    220: // Leak detection
      IF TRUE
      AND _m_LeakTest1_LeakDet()
			THEN 
        THIS^.stSeqCtrlGeneral.iInternalSeqStateCase := 230;
			END_IF
      
    230: // Stop and delay
      IF TRUE
      AND _m_Delay(DelayTime:= REAL_TO_TIME(THIS^.stLT1Params.rRestDelay * 1000))
      AND THIS^.itfCounterCyl.M_Stop()
			THEN 
        IF THIS^.bDoubleActing THEN
          THIS^.stSeqCtrlGeneral.iInternalSeqStateCase := 240; 
        ELSE
          THIS^.stSeqCtrlGeneral.iInternalSeqStateCase := 241; 
        END_IF
			END_IF
      
    240: // Move to Middle position
      IF TRUE
      AND THIS^.itfTestCyl.M_ToHP(ePressureType:= E_PRESSURE_TYPE.FORCE, 
                                  rWorkPressure:= THIS^.stLT1Params.rLoadForceB * 1000, 
                                  bPressureRegulation:= FALSE,
                                  eSpeedType:= E_SPEED_TYPE.PERCENT, 
                                  rSpeed:= 50)
      AND THIS^.itfCounterCyl.M_ToHP(ePressureType:= E_PRESSURE_TYPE.VALUE, 
                                     rWorkPressure:= 0, 
                                     bPressureRegulation:= FALSE,
                                     eSpeedType:= E_SPEED_TYPE.PERCENT, 
                                     rSpeed:= 50)
			THEN 
        IF THIS^.itfTestCyl.P_Position <= THIS^.itfTestCyl.P_StrokeLength / 2 THEN
				  THIS^.stSeqCtrlGeneral.iInternalSeqStateCase := 250; 
        END_IF
			END_IF
      
    241: // Move to Middle position
      IF TRUE
      AND THIS^.itfTestCyl.M_ToHP(ePressureType:= E_PRESSURE_TYPE.VALUE, 
                                  rWorkPressure:= 0, 
                                  bPressureRegulation:= FALSE,
                                  eSpeedType:= E_SPEED_TYPE.PERCENT, 
                                  rSpeed:= 50)
      AND THIS^.itfCounterCyl.M_ToWP(ePressureType:= E_PRESSURE_TYPE.FORCE, 
                                     rWorkPressure:= THIS^.stLT1Params.rLoadForceA * 1000, 
                                     bPressureRegulation:= FALSE,
                                     eSpeedType:= E_SPEED_TYPE.PERCENT, 
                                     rSpeed:= 50)
			THEN 
        IF THIS^.itfTestCyl.P_Position <= THIS^.itfTestCyl.P_StrokeLength / 2 THEN
				  THIS^.stSeqCtrlGeneral.iInternalSeqStateCase := 250; 
        END_IF
			END_IF
      
    250: // Stop and lock
      IF TRUE
      AND _m_Delay(DelayTime:= T#1S)
      AND THIS^.itfTestCyl.M_StopAndLock()
      AND THIS^.itfCounterCyl.M_Stop()
			THEN 
        THIS^.stSeqCtrlGeneral.iInternalSeqStateCase := 260; 
			END_IF
      
    260: // Set cylinder pressure to 0
      IF TRUE
      AND THIS^.itfTestCyl.M_SetWorkPressureZero()
			THEN 
        THIS^.stSeqCtrlGeneral.iInternalSeqStateCase := 270; 
			END_IF
      
    270: // Start leak test push (Middle position)
      IF TRUE
      AND _m_Delay(DelayTime:= T#1S)
      AND THIS^.itfCounterCyl.M_ToWP(ePressureType:= E_PRESSURE_TYPE.FORCE, 
                                     rWorkPressure:= THIS^.stLT1Params.rLoadForceA * 1000, 
                                     bPressureRegulation:= TRUE,
                                     eSpeedType:= E_SPEED_TYPE.PERCENT, 
                                     rSpeed:= 100)
			THEN 
        THIS^.stSeqCtrlGeneral.iInternalSeqStateCase := 280;
			END_IF
      
    280: // Leak detection
      IF TRUE
      AND _m_LeakTest1_LeakDet()
			THEN 
        THIS^.stSeqCtrlGeneral.iInternalSeqStateCase := 290;
			END_IF
      
    290: // Stop and delay
      IF TRUE
      AND _m_Delay(DelayTime:= REAL_TO_TIME(THIS^.stLT1Params.rRestDelay * 1000))
      AND THIS^.itfCounterCyl.M_Stop()
			THEN
        IF THIS^.bDoubleActing THEN
          THIS^.stSeqCtrlGeneral.iInternalSeqStateCase := 300; 
        ELSE
          THIS^.stSeqCtrlGeneral.iInternalSeqStateCase := 1000; 
        END_IF 
			END_IF
      
    300: // Start leak test pull (Middle position)
      IF TRUE
      AND _m_Delay(DelayTime:= T#1S)
      AND THIS^.itfCounterCyl.M_ToHP(ePressureType:= E_PRESSURE_TYPE.FORCE, 
                                     rWorkPressure:= THIS^.stLT1Params.rLoadForceB * 1000, 
                                     bPressureRegulation:= TRUE,
                                     eSpeedType:= E_SPEED_TYPE.PERCENT, 
                                     rSpeed:= 100)
			THEN 
        THIS^.stSeqCtrlGeneral.iInternalSeqStateCase := 310;
			END_IF
      
    310: // Leak detection
      IF TRUE
      AND _m_LeakTest1_LeakDet()
			THEN 
        THIS^.stSeqCtrlGeneral.iInternalSeqStateCase := 320;
			END_IF
      
    320: // Stop and delay
      IF TRUE
      AND _m_Delay(DelayTime:= T#5S)
      AND THIS^.itfCounterCyl.M_Stop()
			THEN 
        THIS^.stSeqCtrlGeneral.iInternalSeqStateCase := 1000; 
			END_IF
      
    1000: // Exit seq - Disable low pressure circuit
      IF TRUE
      AND _m_Delay(DelayTime:= T#1S)
      AND THIS^.itfCounterCyl.M_LowPressureCircuit(bAdd:= FALSE)
			THEN 
				THIS^.stSeqCtrlGeneral.iInternalSeqStateCase := 1010;
			END_IF
      
    1010: // Exit seq - Stop
      IF TRUE
      AND _m_Delay(DelayTime:= T#1S) 
      AND THIS^.itfTestCyl.M_StopAndLock()
      AND THIS^.itfCounterCyl.M_Stop()
			THEN 
				THIS^.stSeqCtrlGeneral.iInternalSeqStateCase := 1020;
			END_IF
      
    1020: // Set pressure
      IF TRUE 
			AND THIS^.itfCounterCyl.M_SetWorkPressureZero()
      AND THIS^.itfTestCyl.M_SetWorkPressureZero()
			THEN 
				THIS^.stSeqCtrlGeneral.iInternalSeqStateCase := 9999; 
			END_IF
      
	ELSE
		THIS^.stSeqCtrlGeneral.eActiveSeqState := E_SEQ_GENERAL.DONE;  
	END_CASE
	THIS^.stSeqCtrlGeneral.strExtraInfo := CONCAT('Internal state: ', TO_STRING(THIS^.stSeqCtrlGeneral.iInternalSeqStateCase));
E_SEQ_GENERAL.DONE:;
E_SEQ_GENERAL.ERROR:;
E_SEQ_GENERAL.TIME_OUT:; 

IF TRUE
AND THIS^.stSeqCtrlGeneral.bTimeOutActiveQuit 
THEN
  THIS^.stSeqCtrlGeneral.strExtraInfo := 'Bitte quittieren und erneut testen';
  IF TRUE
  //AND itfOpMode.P_QUIT
  THEN
    THIS^.stSeqCtrlGeneral.eActiveSeqState := E_SEQ_GENERAL.EXECUTE;
	END_IF
  
END_IF

ELSE
  THIS^.stSeqCtrlGeneral.eActiveSeqState := E_SEQ_GENERAL.ERROR;
END_CASE
END_METHOD

METHOD PRIVATE _m_Seq_LEAK_TEST_2 : E_SEQ_PROCESS
VAR_INPUT
END_VAR
VAR
  ActiveSeq: STRING;
END_VAR
//THIS^._m_GeneralStepSetting(StepType:=E_STEP_STATE_TYPE.INIT,
ActiveSeq := TO_STRING(THIS^.eSeq);

CASE THIS^.stSeqCtrlGeneral.eActiveSeqState OF
E_SEQ_GENERAL.READY:;

	
E_SEQ_GENERAL.EXECUTE:;
	IF TRUE
	AND _m_Delay(T#1S)
	THEN
		THIS^.stSeqCtrlGeneral.eActiveSeqState := E_SEQ_GENERAL.RESET;
	END_IF
  
E_SEQ_GENERAL.RESET:;
	stSeqCtrlGeneral.iInternalSeqStateCase := 0;
	IF TRUE
	THEN
		THIS^.stSeqCtrlGeneral.eActiveSeqState := E_SEQ_GENERAL.BUSY;
	END_IF
  
E_SEQ_GENERAL.BUSY:;
	CASE THIS^.stSeqCtrlGeneral.iInternalSeqStateCase OF
		0: // Check if enable
      IF TRUE
      AND THIS^.bEnable 
      AND THIS^.bDoubleActing
      THEN
        THIS^.stSeqCtrlGeneral.iInternalSeqStateCase := 10; 
      ELSE
        THIS^.stSeqCtrlGeneral.iInternalSeqStateCase := 9999; 
			END_IF

    10: // Disable low pressure mode
      IF TRUE 
			AND THIS^.itfTestCyl.M_LowPressureMode(bSet:= FALSE, ePressureType:= E_PRESSURE_TYPE.VALUE, rWorkPressure:= 0)
			THEN 
				THIS^.stSeqCtrlGeneral.iInternalSeqStateCase := 20; 
			END_IF
      
    20: // Disable low pressure mode
      IF TRUE 
			//AND THIS^.itfTestCyl.M_OpenReservoir(bOpenA:= TRUE, bOpenB:= TRUE)
			THEN 
				THIS^.stSeqCtrlGeneral.iInternalSeqStateCase := 30; 
			END_IF
      
    30: // Disable pump 2
      IF TRUE 
			AND THIS^.itfTestCyl.M_Pump2Add(bAdd:= FALSE)
      AND THIS^.itfPump2Pressure.M_SetLimit(ePressureType:= E_PRESSURE_TYPE.PERCENT, rLimit:= 0)
			THEN
        THIS^.stSeqCtrlGeneral.iInternalSeqStateCase := 40; 
			END_IF
      
    40: // Disable pump 3
      IF TRUE 
			AND THIS^.itfTestCyl.M_Pump3Add(bAdd:= FALSE)
      AND THIS^.itfPump3Pressure.M_SetLimit(ePressureType:= E_PRESSURE_TYPE.PERCENT, rLimit:= 0)
			THEN
        THIS^.stSeqCtrlGeneral.iInternalSeqStateCase := 50; 
			END_IF
      
    50: // Disable pump 4
      IF TRUE 
			AND THIS^.itfTestCyl.M_Pump4Add(bAdd:= FALSE)
      AND THIS^.itfPump4Pressure.M_SetLimit(ePressureType:= E_PRESSURE_TYPE.PERCENT, rLimit:= 0)
			THEN
        THIS^.stSeqCtrlGeneral.iInternalSeqStateCase := 60; 
			END_IF
      
    60: // Shut off low pressure circuit to counter cylinder and switch off pump
      IF TRUE 
			AND THIS^.itfCounterCyl.M_LowPressureCircuit(bAdd:= FALSE)
			THEN 
        THIS^.stSeqCtrlGeneral.iInternalSeqStateCase := 70;
			END_IF
      
    70: // Move to HP (Min position)
      IF TRUE
      AND THIS^.itfTestCyl.M_ToHP(ePressureType:= E_PRESSURE_TYPE.FORCE, 
                                  rWorkPressure:= THIS^.stLT2Params.rLoadForceB * 1000, 
                                  bPressureRegulation:= FALSE,
                                  eSpeedType:= E_SPEED_TYPE.PERCENT, 
                                  rSpeed:= 50)
			THEN 
        IF THIS^.itfTestCyl.P_Position <= 0.1 THEN
				  THIS^.stSeqCtrlGeneral.iInternalSeqStateCase := 71; 
        END_IF
			END_IF
      
    71: // Move to HP (Min position)
      IF TRUE
      AND _m_Delay(DelayTime:= T#25S)
      AND THIS^.itfTestCyl.M_Stop()
      AND THIS^.itfCounterCyl.M_ToHP(ePressureType:= E_PRESSURE_TYPE.BAR, 
                                     rWorkPressure:= 10, 
                                     bPressureRegulation:= FALSE,
                                     eSpeedType:= E_SPEED_TYPE.PERCENT, 
                                     rSpeed:= 100)
			THEN 
        THIS^.stSeqCtrlGeneral.iInternalSeqStateCase := 80; 
			END_IF
      
    80: // Stop and lock
      IF TRUE
      AND _m_Delay(DelayTime:= T#3S)
      AND THIS^.itfTestCyl.M_Stop()
      AND THIS^.itfCounterCyl.M_Stop()
			THEN 
        THIS^.stSeqCtrlGeneral.iInternalSeqStateCase := 90; 
			END_IF
      
    90: // Set cylinder pressure to 0
      IF TRUE
      AND THIS^.itfCounterCyl.M_SetWorkPressureZero()
      AND THIS^.itfTestCyl.M_OpenReservoir(bOpenA:= TRUE, bOpenB:= FALSE)
			THEN 
        THIS^.stSeqCtrlGeneral.iInternalSeqStateCase := 100; 
			END_IF
      
    100: // Start leak test push (HP endposition)
      IF TRUE
      AND _m_Delay(DelayTime:= T#1S)
      AND THIS^.itfTestCyl.M_ToHP(ePressureType:= E_PRESSURE_TYPE.FORCE, 
                                  rWorkPressure:= THIS^.stLT2Params.rLoadForceB * 1000, 
                                  bPressureRegulation:= TRUE,
                                  eSpeedType:= E_SPEED_TYPE.PERCENT, 
                                  rSpeed:= 100)
			THEN 
        THIS^.stSeqCtrlGeneral.iInternalSeqStateCase := 110;
			END_IF
      
    110: // Set lock valves
      IF TRUE
      AND _m_Delay(DelayTime:= T#1S)
      AND THIS^.itfTestCyl.M_OpenLockValves(bOpenChA:= FALSE, bOpenChB:= TRUE)
			THEN 
        THIS^.stSeqCtrlGeneral.iInternalSeqStateCase := 120;
			END_IF
      
    120: // Leak detection
      THIS^.siLT2TestDirection := -1;
      IF TRUE
      AND _m_LeakTest2_LeakDet()
			THEN 
        THIS^.stSeqCtrlGeneral.iInternalSeqStateCase := 130;
			END_IF
      
    130: // Stop and delay
      IF TRUE
      AND _m_Delay(DelayTime:= REAL_TO_TIME(THIS^.stLT2Params.rRestDelay * 1000))
      AND THIS^.itfTestCyl.M_Stop()
			THEN 
        THIS^.stSeqCtrlGeneral.iInternalSeqStateCase := 140; 
			END_IF
      
    140: // Move to WP (Max position)
      IF TRUE
      AND THIS^.itfTestCyl.M_ToWP(ePressureType:= E_PRESSURE_TYPE.FORCE, 
                                  rWorkPressure:= THIS^.stLT2Params.rLoadForceA * 1000, 
                                  bPressureRegulation:= FALSE,
                                  eSpeedType:= E_SPEED_TYPE.PERCENT, 
                                  rSpeed:= 50)
			THEN 
        IF THIS^.itfTestCyl.P_Position >= THIS^.itfTestCyl.P_StrokeLength - 0.1 THEN
				  THIS^.stSeqCtrlGeneral.iInternalSeqStateCase := 150; 
        END_IF
			END_IF
      
    150: // Stop and lock
      IF TRUE
      AND _m_Delay(DelayTime:= T#3S)
      AND THIS^.itfTestCyl.M_Stop()
      AND THIS^.itfCounterCyl.M_Stop()
			THEN 
        THIS^.stSeqCtrlGeneral.iInternalSeqStateCase := 160; 
			END_IF
      
    160: // Set cylinder pressure to 0
      IF TRUE
      AND THIS^.itfCounterCyl.M_SetWorkPressureZero()
      AND THIS^.itfTestCyl.M_OpenReservoir(bOpenA:= FALSE, bOpenB:= TRUE)
			THEN 
        THIS^.stSeqCtrlGeneral.iInternalSeqStateCase := 170; 
			END_IF
      
    170: // Start leak test push (WP endposition)
      IF TRUE
      AND _m_Delay(DelayTime:= T#1S)
      AND THIS^.itfTestCyl.M_ToWP(ePressureType:= E_PRESSURE_TYPE.FORCE, 
                                  rWorkPressure:= THIS^.stLT2Params.rLoadForceA * 1000, 
                                  bPressureRegulation:= TRUE,
                                  eSpeedType:= E_SPEED_TYPE.PERCENT, 
                                  rSpeed:= 100)
			THEN 
        THIS^.stSeqCtrlGeneral.iInternalSeqStateCase := 180;
			END_IF
      
    180: // Set lock valves
      IF TRUE
      AND _m_Delay(DelayTime:= T#1S)
      AND THIS^.itfTestCyl.M_OpenLockValves(bOpenChA:= TRUE, bOpenChB:= FALSE)
			THEN 
        THIS^.stSeqCtrlGeneral.iInternalSeqStateCase := 190;
			END_IF
      
    190: // Leak detection
      THIS^.siLT2TestDirection := 1;
      IF TRUE
      AND _m_LeakTest2_LeakDet()
			THEN 
        THIS^.stSeqCtrlGeneral.iInternalSeqStateCase := 200;
			END_IF
      
    200: // Stop and delay
      IF TRUE
      AND _m_Delay(DelayTime:= T#1S)
      AND THIS^.itfTestCyl.M_Stop()
			THEN 
        THIS^.stSeqCtrlGeneral.iInternalSeqStateCase := 1000; 
			END_IF
      
    1000: // Exit seq - Disable low pressure circuit
      IF TRUE
      AND _m_Delay(DelayTime:= T#1S)
      AND THIS^.itfCounterCyl.M_LowPressureCircuit(bAdd:= FALSE)
			THEN 
				THIS^.stSeqCtrlGeneral.iInternalSeqStateCase := 1010;
			END_IF
      
    1010: // Exit seq - Stop
      IF TRUE
      AND _m_Delay(DelayTime:= T#1S) 
      AND THIS^.itfTestCyl.M_StopAndLock()
      AND THIS^.itfCounterCyl.M_Stop()
			THEN 
				THIS^.stSeqCtrlGeneral.iInternalSeqStateCase := 1020;
			END_IF
      
    1020: // Set pressure
      IF TRUE 
			AND THIS^.itfCounterCyl.M_SetWorkPressureZero()
      AND THIS^.itfTestCyl.M_SetWorkPressureZero()
			THEN 
				THIS^.stSeqCtrlGeneral.iInternalSeqStateCase := 1030; 
			END_IF
      
    1030: // Disable reservoir
      IF TRUE 
      AND THIS^.itfTestCyl.M_OpenReservoir(bOpenA:= FALSE, bOpenB:= FALSE)
			THEN 
				THIS^.stSeqCtrlGeneral.iInternalSeqStateCase := 9999; 
			END_IF
      
	ELSE
		THIS^.stSeqCtrlGeneral.eActiveSeqState := E_SEQ_GENERAL.DONE;  
	END_CASE
	THIS^.stSeqCtrlGeneral.strExtraInfo := CONCAT('Internal state: ', TO_STRING(THIS^.stSeqCtrlGeneral.iInternalSeqStateCase));
E_SEQ_GENERAL.DONE:;
E_SEQ_GENERAL.ERROR:;
E_SEQ_GENERAL.TIME_OUT:; 

IF TRUE
AND THIS^.stSeqCtrlGeneral.bTimeOutActiveQuit 
THEN
  THIS^.stSeqCtrlGeneral.strExtraInfo := 'Bitte quittieren und erneut testen';
  IF TRUE
  //AND itfOpMode.P_QUIT
  THEN
    THIS^.stSeqCtrlGeneral.eActiveSeqState := E_SEQ_GENERAL.EXECUTE;
	END_IF
  
END_IF

ELSE
  THIS^.stSeqCtrlGeneral.eActiveSeqState := E_SEQ_GENERAL.ERROR;
END_CASE
END_METHOD

METHOD PRIVATE _m_Seq_MAX_SPEED_RECORD : E_SEQ_PROCESS
VAR_INPUT
END_VAR
VAR
  ActiveSeq:            STRING;
END_VAR
//THIS^._m_GeneralStepSetting(StepType:=E_STEP_STATE_TYPE.INIT,
ActiveSeq := TO_STRING(THIS^.eSeq);

// Distance record
_m_DistanceRecord();

CASE THIS^.stSeqCtrlGeneral.eActiveSeqState OF
E_SEQ_GENERAL.READY:;

	
E_SEQ_GENERAL.EXECUTE:;
	IF TRUE
	AND _m_Delay(T#1S)
	THEN
		THIS^.stSeqCtrlGeneral.eActiveSeqState := E_SEQ_GENERAL.RESET;
	END_IF
  
E_SEQ_GENERAL.RESET:;
	stSeqCtrlGeneral.iInternalSeqStateCase := 0;
	IF TRUE
	THEN
    THIS^.udiCurrentCycle := 1;
    THIS^.lrTotalSpeed := 0.0;
    THIS^.udiSpeedDividend := 0;
		THIS^.stSeqCtrlGeneral.eActiveSeqState := E_SEQ_GENERAL.BUSY;
	END_IF
  
E_SEQ_GENERAL.BUSY:;
	CASE THIS^.stSeqCtrlGeneral.iInternalSeqStateCase OF
    0: // Check if enable
      IF TRUE
      AND THIS^.bEnable 
      AND THIS^.itfTestCyl.P_StrokeLength - 60 > 50
      THEN
        THIS^.stSeqCtrlGeneral.iInternalSeqStateCase := 10; 
      ELSE
        THIS^.stSeqCtrlGeneral.iInternalSeqStateCase := 9999; 
			END_IF
    
		10: // Disable low pressure mode
      IF TRUE 
			AND THIS^.itfTestCyl.M_LowPressureMode(bSet:= FALSE, ePressureType:= E_PRESSURE_TYPE.VALUE, rWorkPressure:= 0)
			THEN
        THIS^.stSeqCtrlGeneral.iInternalSeqStateCase := 20;
			END_IF
      
    20: // Add low pressure circuit to counter cylinder
      IF TRUE 
			AND THIS^.itfCounterCyl.M_LowPressureCircuit(bAdd:= TRUE)
			THEN 
				THIS^.stSeqCtrlGeneral.iInternalSeqStateCase := 30; 
			END_IF
      
    30: // Move to HP (Min position + 10)
      IF TRUE
      AND THIS^.itfTestCyl.M_ToHP(ePressureType:= E_PRESSURE_TYPE.FORCE, 
                                  rWorkPressure:= THIS^.stERParams.rWorkForceB * 1000, 
                                  bPressureRegulation:= TRUE,
                                  eSpeedType:= E_SPEED_TYPE.PERCENT, 
                                  rSpeed:= 100)
			THEN 
        IF THIS^.bDoubleActing THEN
          THIS^.stSeqCtrlGeneral.iInternalSeqStateCase := 31;
        ELSE
          THIS^.stSeqCtrlGeneral.iInternalSeqStateCase := 32;
        END_IF
			END_IF
      
    31: // Move to HP (Min position + 10)
      IF TRUE
      AND THIS^.itfCounterCyl.M_ToHP( ePressureType:= E_PRESSURE_TYPE.FORCE, 
                                      rWorkPressure:= THIS^.stERParams.rLoadForceB * 1000, 
                                      bPressureRegulation:= TRUE,
                                      eSpeedType:= E_SPEED_TYPE.PERCENT, 
                                      rSpeed:= 100)
			THEN 
        THIS^.stSeqCtrlGeneral.iInternalSeqStateCase := 40;
			END_IF
      
    32: // Move to HP (Min position + 10)
      IF TRUE
      AND THIS^.itfCounterCyl.M_ToWP( ePressureType:= E_PRESSURE_TYPE.FORCE, 
                                      rWorkPressure:= THIS^.stERParams.rLoadForceA * 1000, 
                                      bPressureRegulation:= FALSE,
                                      eSpeedType:= E_SPEED_TYPE.PERCENT, 
                                      rSpeed:= 100)
			THEN 
        THIS^.stSeqCtrlGeneral.iInternalSeqStateCase := 40;
			END_IF
      
    40: // Move to HP (Min position + 10)
      IF TRUE
			THEN 
        IF THIS^.itfTestCyl.P_Position <= ABS(THIS^.stERParams.rTurningPointHP) THEN
				  THIS^.stSeqCtrlGeneral.iInternalSeqStateCase := 50;
        END_IF
			END_IF
      
    50: // Stop
      IF TRUE
      AND _m_Delay(DelayTime:= T#1S)
      AND THIS^.itfTestCyl.M_Stop()
      AND THIS^.itfCounterCyl.M_Stop()
			THEN 
        THIS^.stSeqCtrlGeneral.iInternalSeqStateCase := 55; 
			END_IF

    55: // Choice step
      IF TRUE 
			THEN 
        IF TRUE
        AND THIS^.udiCurrentCycle > 3 
        THEN
          THIS^.stSeqCtrlGeneral.iInternalSeqStateCase := 100; // Save and exit
        ELSE
          THIS^.stSeqCtrlGeneral.iInternalSeqStateCase := 60; 
				END_IF
			END_IF
      
    60: // Stop
      IF TRUE
      AND _m_Delay(DelayTime:= T#1S)
      AND THIS^.itfTestCyl.M_Stop()
      AND THIS^.itfCounterCyl.M_Stop()
			THEN 
        THIS^.stSeqCtrlGeneral.iInternalSeqStateCase := 70; 
			END_IF
      
    70: // Move to WP (Max position - 10)
      IF TRUE
      AND THIS^.itfTestCyl.M_ToWP(ePressureType:= E_PRESSURE_TYPE.FORCE, 
                                  rWorkPressure:= THIS^.stERParams.rWorkForceA * 1000, 
                                  bPressureRegulation:= TRUE,
                                  eSpeedType:= E_SPEED_TYPE.PERCENT, 
                                  rSpeed:= 100)
			THEN 
        THIS^.stSeqCtrlGeneral.iInternalSeqStateCase := 71;
			END_IF
      
    71: // Move to WP (Max position - 10)
      IF TRUE
      AND THIS^.itfCounterCyl.M_ToWP( ePressureType:= E_PRESSURE_TYPE.FORCE, 
                                      rWorkPressure:= THIS^.stERParams.rLoadForceA * 1000, 
                                      bPressureRegulation:= TRUE,
                                      eSpeedType:= E_SPEED_TYPE.PERCENT, 
                                      rSpeed:= 100)
			THEN 
        IF THIS^.itfTestCyl.P_Position >= 30 THEN
				  THIS^.stSeqCtrlGeneral.iInternalSeqStateCase := 72; 
        END_IF
			END_IF
      
    72: // Start record
      IF TRUE
      AND THIS^.itfTestCyl.P_Position <= THIS^.itfTestCyl.P_StrokeLength - 30
			THEN 
        THIS^.lrTotalSpeed := THIS^.lrTotalSpeed + ABS(THIS^.itfTestCyl.P_SpeedInMmPerSecond);
        THIS^.udiSpeedDividend := THIS^.udiSpeedDividend + 1;
      ELSE
        THIS^.listSpeed[THIS^.udiCurrentCycle] := THIS^.lrTotalSpeed / THIS^.udiSpeedDividend;
        THIS^.lrTotalSpeed := 0.0;
        THIS^.udiSpeedDividend := 0;
        THIS^.stSeqCtrlGeneral.iInternalSeqStateCase := 73;
			END_IF
      
    73: // Move to WP (Max position - 10)
      IF TRUE
      AND THIS^.itfTestCyl.P_Position >= THIS^.itfTestCyl.P_StrokeLength - ABS(THIS^.stERParams.rTurningPointWP) THEN
				THIS^.stSeqCtrlGeneral.iInternalSeqStateCase := 80;
			END_IF
      
    80: // Stop
      IF TRUE
      AND _m_Delay(DelayTime:= T#1S)
      AND THIS^.itfTestCyl.M_Stop()
      AND THIS^.itfCounterCyl.M_Stop()
			THEN 
        THIS^.stSeqCtrlGeneral.iInternalSeqStateCase := 90; 
			END_IF
      
    90: // Move to HP (Min position + 10)
      IF TRUE
      AND THIS^.itfTestCyl.M_ToHP(ePressureType:= E_PRESSURE_TYPE.FORCE, 
                                  rWorkPressure:= THIS^.stERParams.rWorkForceB * 1000, 
                                  bPressureRegulation:= TRUE,
                                  eSpeedType:= E_SPEED_TYPE.PERCENT, 
                                  rSpeed:= 100)
			THEN 
        IF THIS^.bDoubleActing THEN
          THIS^.stSeqCtrlGeneral.iInternalSeqStateCase := 91;
        ELSE
          THIS^.stSeqCtrlGeneral.iInternalSeqStateCase := 92;
        END_IF
			END_IF
      
    91: // Move to HP (Min position + 10)
      IF TRUE
      AND THIS^.itfCounterCyl.M_ToHP( ePressureType:= E_PRESSURE_TYPE.FORCE, 
                                      rWorkPressure:= THIS^.stERParams.rLoadForceB * 1000, 
                                      bPressureRegulation:= TRUE,
                                      eSpeedType:= E_SPEED_TYPE.PERCENT, 
                                      rSpeed:= 100)
			THEN 
        IF THIS^.itfTestCyl.P_Position <= THIS^.itfTestCyl.P_StrokeLength - 30 THEN
				  THIS^.stSeqCtrlGeneral.iInternalSeqStateCase := 95;
        END_IF
			END_IF
      
    92: // Move to HP (Min position + 10)
      IF TRUE
      AND THIS^.itfCounterCyl.M_ToWP( ePressureType:= E_PRESSURE_TYPE.FORCE, 
                                      rWorkPressure:= THIS^.stERParams.rLoadForceB * 1000, 
                                      bPressureRegulation:= FALSE,
                                      eSpeedType:= E_SPEED_TYPE.PERCENT, 
                                      rSpeed:= 100)
			THEN 
        IF THIS^.itfTestCyl.P_Position <= THIS^.itfTestCyl.P_StrokeLength - 30 THEN
				  THIS^.stSeqCtrlGeneral.iInternalSeqStateCase := 95;
        END_IF
			END_IF
      
    95: // Start record
      IF TRUE
      AND THIS^.itfTestCyl.P_Position >= 30
			THEN 
        THIS^.lrTotalSpeed := THIS^.lrTotalSpeed + ABS(THIS^.itfTestCyl.P_SpeedInMmPerSecond);
        THIS^.udiSpeedDividend := THIS^.udiSpeedDividend + 1;
      ELSE
        THIS^.listSpeed[THIS^.udiCurrentCycle + 3] := THIS^.lrTotalSpeed / THIS^.udiSpeedDividend;
        THIS^.lrTotalSpeed := 0.0;
        THIS^.udiSpeedDividend := 0;
        THIS^.stSeqCtrlGeneral.iInternalSeqStateCase := 96;
			END_IF
      
    96: // Move to HP (Min position + 10)
      IF TRUE
      AND THIS^.itfTestCyl.P_Position <= ABS(THIS^.stERParams.rTurningPointHP) THEN
        THIS^.udiCurrentCycle := THIS^.udiCurrentCycle + 1;
				THIS^.stSeqCtrlGeneral.iInternalSeqStateCase := 55; // Jump backward
			END_IF
      
    100: // Set max speed
      IF TRUE
      THEN
        FOR THIS^.ii := 1 TO 3 BY 1 DO
          IF THIS^.ii = 1 THEN
            IF THIS^.bDoubleActing THEN
              THIS^.rMaxSpeedInMmPerSHP := THIS^.listSpeed[THIS^.ii + 3];
            END_IF
            THIS^.rMaxSpeedInMmPerSWP := THIS^.listSpeed[THIS^.ii];
          ELSE
            IF THIS^.rMaxSpeedInMmPerSHP > THIS^.listSpeed[THIS^.ii + 3] AND THIS^.bDoubleActing THEN
              THIS^.rMaxSpeedInMmPerSHP := THIS^.listSpeed[THIS^.ii + 3];
						END_IF
            IF THIS^.rMaxSpeedInMmPerSWP > THIS^.listSpeed[THIS^.ii] THEN
              THIS^.rMaxSpeedInMmPerSWP := THIS^.listSpeed[THIS^.ii];
						END_IF
					END_IF
        END_FOR  
        IF THIS^.ii >= 3 THEN
          THIS^.ii := 1;
          THIS^.stSeqCtrlGeneral.iInternalSeqStateCase := 1000;
				END_IF
			END_IF
      
    1000: // Exit seq - Disable low pressure circuit
      IF TRUE
      AND _m_Delay(DelayTime:= T#1S)
      AND THIS^.itfCounterCyl.M_LowPressureCircuit(bAdd:= FALSE)
			THEN 
				THIS^.stSeqCtrlGeneral.iInternalSeqStateCase := 1010;
			END_IF  
      
    1010: // Exit seq - Stop
      IF TRUE
      AND _m_Delay(DelayTime:= T#1S) 
      AND THIS^.itfTestCyl.M_StopAndLock()
      AND THIS^.itfCounterCyl.M_Stop()
			THEN 
				THIS^.stSeqCtrlGeneral.iInternalSeqStateCase := 1020;
			END_IF
      
    1020: // Set pressure
      IF TRUE 
			AND THIS^.itfCounterCyl.M_SetWorkPressureZero()
      AND THIS^.itfTestCyl.M_SetWorkPressureZero()
			THEN 
				THIS^.stSeqCtrlGeneral.iInternalSeqStateCase := 1030; 
			END_IF
      
    1030: // Remove pump 2
      IF TRUE 
			AND THIS^.itfTestCyl.M_Pump2Add(bAdd:= FALSE)
      //AND THIS^.itfPump2Pressure.M_SetLimit(ePressureType:= E_PRESSURE_TYPE.PERCENT, rLimit:= 0)
			THEN
        THIS^.stSeqCtrlGeneral.iInternalSeqStateCase := 1040; 
			END_IF
      
    1040: // Remove pump 3
      IF TRUE 
			AND THIS^.itfTestCyl.M_Pump3Add(bAdd:= FALSE)
      //AND THIS^.itfPump3Pressure.M_SetLimit(ePressureType:= E_PRESSURE_TYPE.PERCENT, rLimit:= 0)
			THEN
        THIS^.stSeqCtrlGeneral.iInternalSeqStateCase := 1050; 
			END_IF
      
    1050: // Remove pump 4
      IF TRUE 
			AND THIS^.itfTestCyl.M_Pump4Add(bAdd:= FALSE)
      //AND THIS^.itfPump4Pressure.M_SetLimit(ePressureType:= E_PRESSURE_TYPE.PERCENT, rLimit:= 0)
			THEN
        THIS^.stSeqCtrlGeneral.iInternalSeqStateCase := 9999; 
			END_IF
      
	ELSE
		THIS^.stSeqCtrlGeneral.eActiveSeqState := E_SEQ_GENERAL.DONE;  
	END_CASE
	THIS^.stSeqCtrlGeneral.strExtraInfo := CONCAT('Internal state: ', TO_STRING(THIS^.stSeqCtrlGeneral.iInternalSeqStateCase));

E_SEQ_GENERAL.DONE:;
E_SEQ_GENERAL.ERROR:;
E_SEQ_GENERAL.TIME_OUT:; 

IF TRUE
AND THIS^.stSeqCtrlGeneral.bTimeOutActiveQuit 
THEN
  THIS^.stSeqCtrlGeneral.strExtraInfo := 'Bitte quittieren und erneut testen';
  IF TRUE
  //AND itfOpMode.P_QUIT
  THEN
    THIS^.stSeqCtrlGeneral.eActiveSeqState := E_SEQ_GENERAL.EXECUTE;
	END_IF
  
END_IF

ELSE
  THIS^.stSeqCtrlGeneral.eActiveSeqState := E_SEQ_GENERAL.ERROR;
END_CASE
END_METHOD

METHOD PRIVATE _m_Seq_MEASURE_STROKE_LENGTH : E_SEQ_PROCESS
VAR_INPUT
END_VAR
VAR
  ActiveSeq: STRING;
END_VAR
//THIS^._m_GeneralStepSetting(StepType:=E_STEP_STATE_TYPE.INIT,
ActiveSeq := TO_STRING(THIS^.eSeq);

// Distance record
_m_DistanceRecord();

CASE THIS^.stSeqCtrlGeneral.eActiveSeqState OF
E_SEQ_GENERAL.READY:;
	
E_SEQ_GENERAL.EXECUTE:;
	IF TRUE
	AND _m_Delay(T#1S)
	THEN
		THIS^.stSeqCtrlGeneral.eActiveSeqState := E_SEQ_GENERAL.RESET;
	END_IF
  
E_SEQ_GENERAL.RESET:;
	stSeqCtrlGeneral.iInternalSeqStateCase := 0;
  
	IF TRUE
	THEN
		THIS^.stSeqCtrlGeneral.eActiveSeqState := E_SEQ_GENERAL.BUSY;
	END_IF
  
E_SEQ_GENERAL.BUSY:;
	CASE THIS^.stSeqCtrlGeneral.iInternalSeqStateCase OF
		0: // Check if enable
      IF TRUE
      AND THIS^.bEnable 
      THEN
        THIS^.stSeqCtrlGeneral.iInternalSeqStateCase := 10; 
      ELSE
        THIS^.stSeqCtrlGeneral.iInternalSeqStateCase := 9999; 
			END_IF

    10: // Disable low pressure mode and add low pressure to counter cylinder
      IF TRUE 
			AND THIS^.itfTestCyl.M_LowPressureMode(bSet:= FALSE, ePressureType:= E_PRESSURE_TYPE.VALUE, rWorkPressure:= 0)
      AND THIS^.itfCounterCyl.M_LowPressureCircuit(bAdd:= TRUE)
			THEN 
				THIS^.stSeqCtrlGeneral.iInternalSeqStateCase := 20; 
			END_IF
      
    20: // Disable pump 2
      IF TRUE 
			AND THIS^.itfTestCyl.M_Pump2Add(bAdd:= FALSE)
      //AND THIS^.itfPump2Pressure.M_SetLimit(ePressureType:= E_PRESSURE_TYPE.PERCENT, rLimit:= 0)
			THEN
        THIS^.stSeqCtrlGeneral.iInternalSeqStateCase := 30; 
			END_IF
      
    30: // Disable pump 3
      IF TRUE 
			AND THIS^.itfTestCyl.M_Pump3Add(bAdd:= FALSE)
      //AND THIS^.itfPump3Pressure.M_SetLimit(ePressureType:= E_PRESSURE_TYPE.PERCENT, rLimit:= 0)
			THEN
        THIS^.stSeqCtrlGeneral.iInternalSeqStateCase := 40; 
			END_IF
      
    40: // Disable pump 4
      IF TRUE 
			AND THIS^.itfTestCyl.M_Pump4Add(bAdd:= FALSE)
      //AND THIS^.itfPump4Pressure.M_SetLimit(ePressureType:= E_PRESSURE_TYPE.PERCENT, rLimit:= 0)
			THEN
        THIS^.stSeqCtrlGeneral.iInternalSeqStateCase := 50; 
			END_IF
      
    50: // Check if double- or single-acting cylinder
      IF TRUE 
      AND THIS^.bDoubleActing
			THEN 
        THIS^.stSeqCtrlGeneral.iInternalSeqStateCase := 60;
      ELSE
        THIS^.stSeqCtrlGeneral.iInternalSeqStateCase := 61;
			END_IF
      
		60:	// Double acting cylinder - Move to HP
      IF TRUE 
      AND THIS^.itfTestCyl.M_ToHP(ePressureType:= E_PRESSURE_TYPE.FORCE, 
                                  rWorkPressure:= THIS^.rWorkForceBTmp * 1000, 
                                  bPressureRegulation:= FALSE,
                                  eSpeedType:= E_SPEED_TYPE.PERCENT, 
                                  rSpeed:= 50)
      AND THIS^.itfCounterCyl.M_ToHP(ePressureType:= E_PRESSURE_TYPE.VALUE, 
                                      rWorkPressure:= 0, 
                                      bPressureRegulation:= FALSE,
                                      eSpeedType:= E_SPEED_TYPE.PERCENT, 
                                      rSpeed:= 50)
			THEN 
        THIS^.stSeqCtrlGeneral.iInternalSeqStateCase := 70;
			END_IF
      
    61:	// Single acting cylinder - Move to HP
      IF TRUE 
      AND THIS^.itfTestCyl.M_ToHP(ePressureType:= E_PRESSURE_TYPE.VALUE, 
                                  rWorkPressure:= 0, 
                                  bPressureRegulation:= FALSE,
                                  eSpeedType:= E_SPEED_TYPE.PERCENT, 
                                  rSpeed:= 50)
			THEN 
        THIS^.stSeqCtrlGeneral.iInternalSeqStateCase := 62;
			END_IF
      
    62: // Cylinder - Move to HP - Check if Cylinder decoupled
      IF TRUE
      AND NOT THIS^.bCylinderDecoupled
      THEN
        IF THIS^.itfCounterCyl.M_ToWP(ePressureType:= E_PRESSURE_TYPE.FORCE, 
                                      rWorkPressure:= THIS^.rLoadForceATmp * 1000, 
                                      bPressureRegulation:= FALSE,
                                      eSpeedType:= E_SPEED_TYPE.PERCENT, 
                                      rSpeed:= 50)
			  THEN 
          THIS^.stSeqCtrlGeneral.iInternalSeqStateCase := 70;
        END_IF
      ELSE
        THIS^.stSeqCtrlGeneral.iInternalSeqStateCase := 70;
			END_IF
      
    70:	// Delay timer
      IF TRUE 
      AND _m_Delay(DelayTime:= T#3S)
			THEN 
        THIS^.stSeqCtrlGeneral.iInternalSeqStateCase := 71;
			END_IF
      
    71:	// Wait for HP endpos
      IF TRUE 
			THEN 
        IF TRUE 
        AND ABS(THIS^.itfTestCyl.P_PositionAbs - THIS^.lrLastPos) < 0.1
        THEN
          THIS^.stSeqCtrlGeneral.iInternalSeqStateCase := 80;
        ELSE
          THIS^.lrLastPos := THIS^.itfTestCyl.P_PositionAbs;
          THIS^.stSeqCtrlGeneral.iInternalSeqStateCase := 70;
        END_IF
			END_IF
      
    80:	// Set zero position
      IF TRUE 
      AND THIS^.itfTestCyl.M_SetZeroPos()
			THEN 
        THIS^.stSeqCtrlGeneral.iInternalSeqStateCase := 90;
			END_IF
      
    90: // Vent cylinder - Move to WP (Max position)
      IF TRUE
      AND NOT THIS^.bCylinderDecoupled
			THEN 
				THIS^.stSeqCtrlGeneral.iInternalSeqStateCase := 91; 
      ELSE
        THIS^.stSeqCtrlGeneral.iInternalSeqStateCase := 92; 
			END_IF
      
    91:	// Move to WP
      IF TRUE 
      AND THIS^.itfTestCyl.M_ToWP(ePressureType:= E_PRESSURE_TYPE.FORCE, 
                                  rWorkPressure:= THIS^.rWorkForceATmp * 1000, 
                                  bPressureRegulation:= FALSE,
                                  eSpeedType:= E_SPEED_TYPE.PERCENT, 
                                  rSpeed:= 50)
      AND THIS^.itfCounterCyl.M_ToWP(ePressureType:= E_PRESSURE_TYPE.VALUE, 
                                     rWorkPressure:= 0, 
                                     bPressureRegulation:= FALSE,
                                     eSpeedType:= E_SPEED_TYPE.PERCENT, 
                                     rSpeed:= 50)
			THEN 
        THIS^.stSeqCtrlGeneral.iInternalSeqStateCase := 100;
			END_IF
      
    92:	// Move to WP
      IF TRUE 
      AND THIS^.itfTestCyl.M_ToWP(ePressureType:= E_PRESSURE_TYPE.FORCE, 
                                  rWorkPressure:= THIS^.rWorkForceATmp * 1000, 
                                  bPressureRegulation:= FALSE,
                                  eSpeedType:= E_SPEED_TYPE.PERCENT, 
                                  rSpeed:= 50)
      AND THIS^.itfCounterCyl.M_ToHP(ePressureType:= E_PRESSURE_TYPE.VALUE, 
                                     rWorkPressure:= 0, 
                                     bPressureRegulation:= FALSE,
                                     eSpeedType:= E_SPEED_TYPE.PERCENT, 
                                     rSpeed:= 50)
			THEN 
        THIS^.stSeqCtrlGeneral.iInternalSeqStateCase := 100;
			END_IF
      
    100:	// Delay timer
      IF TRUE 
      AND _m_Delay(DelayTime:= T#3S)
			THEN 
        THIS^.stSeqCtrlGeneral.iInternalSeqStateCase := 101;
			END_IF
      
    101:	// Wait for WP endpos
      IF TRUE 
			THEN 
        IF TRUE 
        AND ABS(THIS^.itfTestCyl.P_PositionAbs - THIS^.lrLastPos) < 0.1
        THEN
          THIS^.stSeqCtrlGeneral.iInternalSeqStateCase := 110;
        ELSE
          THIS^.lrLastPos := THIS^.itfTestCyl.P_PositionAbs;
          THIS^.stSeqCtrlGeneral.iInternalSeqStateCase := 100;
        END_IF
			END_IF
      
    110:	// Set Max position
      IF TRUE 
      AND THIS^.itfTestCyl.M_SetMaxPos()
			THEN 
        THIS^.stSeqCtrlGeneral.iInternalSeqStateCase := 120;
			END_IF
      
    120:	// Stop
      IF TRUE 
      AND THIS^.itfCounterCyl.M_Stop()
      AND THIS^.itfTestCyl.M_StopAndLock()
			THEN 
        THIS^.stSeqCtrlGeneral.iInternalSeqStateCase := 130;
			END_IF
      
    130:	// Set work/load pressure
      IF TRUE 
      AND itfTestCyl.M_SetWorkPressureZero()
      AND itfCounterCyl.M_SetWorkPressureZero()
			THEN 
        THIS^.stSeqCtrlGeneral.iInternalSeqStateCase := 140;
			END_IF
      
    140: // Disable low pressure mode
      IF TRUE 
      AND THIS^.itfCounterCyl.M_LowPressureCircuit(bAdd:= FALSE)
			THEN 
				THIS^.stSeqCtrlGeneral.iInternalSeqStateCase := 1000; 
			END_IF
      
    1000: // Exit step
      IF TRUE
			THEN 
				THIS^.stSeqCtrlGeneral.iInternalSeqStateCase := 9999;
			END_IF
      
	ELSE
		THIS^.stSeqCtrlGeneral.eActiveSeqState:=E_SEQ_GENERAL.DONE;  
	END_CASE
	THIS^.stSeqCtrlGeneral.strExtraInfo:=concat('Internal state: ', TO_STRING(THIS^.stSeqCtrlGeneral.iInternalSeqStateCase));
E_SEQ_GENERAL.DONE:;
E_SEQ_GENERAL.ERROR:;
E_SEQ_GENERAL.TIME_OUT:; 

IF TRUE
AND THIS^.stSeqCtrlGeneral.bTimeOutActiveQuit 
THEN
  THIS^.stSeqCtrlGeneral.strExtraInfo:= 'Bitte quittieren und erneut testen';
  IF TRUE
  //AND itfOpMode.P_QUIT
  THEN
    THIS^.stSeqCtrlGeneral.eActiveSeqState:=E_SEQ_GENERAL.EXECUTE;
	END_IF
  
END_IF

ELSE
  THIS^.stSeqCtrlGeneral.eActiveSeqState:=E_SEQ_GENERAL.ERROR;
END_CASE
END_METHOD

METHOD PRIVATE _m_Seq_MOVE_CYL1_TO_HP : E_SEQ_PROCESS
VAR_INPUT
END_VAR
VAR
  ActiveSeq: STRING;
END_VAR
//THIS^._m_GeneralStepSetting(StepType:=E_STEP_STATE_TYPE.INIT,
ActiveSeq := TO_STRING(THIS^.eSeq);

// Distance record
_m_DistanceRecord();

CASE THIS^.stSeqCtrlGeneral.eActiveSeqState OF
E_SEQ_GENERAL.READY:;

E_SEQ_GENERAL.EXECUTE:;
	IF TRUE
	AND _m_Delay(T#1S)
	THEN
		THIS^.stSeqCtrlGeneral.eActiveSeqState := E_SEQ_GENERAL.RESET;
	END_IF
  
E_SEQ_GENERAL.RESET:;
	stSeqCtrlGeneral.iInternalSeqStateCase := 0;
  IF TRUE
	THEN
    THIS^.udiCurrentCycle := 1;
		THIS^.stSeqCtrlGeneral.eActiveSeqState := E_SEQ_GENERAL.BUSY;
	END_IF
  
E_SEQ_GENERAL.BUSY:;
	CASE THIS^.stSeqCtrlGeneral.iInternalSeqStateCase OF
    0: // Check if enable
      IF TRUE
      AND THIS^.bEnable 
      THEN
        THIS^.stSeqCtrlGeneral.iInternalSeqStateCase := 10; 
      ELSE
        THIS^.stSeqCtrlGeneral.iInternalSeqStateCase := 9999; 
			END_IF

    10: // Disable low pressure mode
      IF TRUE 
      AND _m_Delay(DelayTime:= T#3S)
			AND THIS^.itfTestCyl.M_LowPressureMode(bSet:= FALSE, ePressureType:= E_PRESSURE_TYPE.VALUE, rWorkPressure:= 0)
			THEN 
				THIS^.stSeqCtrlGeneral.iInternalSeqStateCase := 20; 
			END_IF
      
    20: // Disable pump 2
      IF TRUE 
			AND THIS^.itfTestCyl.M_Pump2Add(bAdd:= FALSE)
      //AND THIS^.itfPump2Pressure.M_SetLimit(ePressureType:= E_PRESSURE_TYPE.PERCENT, rLimit:= 0)
			THEN
        THIS^.stSeqCtrlGeneral.iInternalSeqStateCase := 30; 
			END_IF
      
    30: // Disable pump 3
      IF TRUE 
			AND THIS^.itfTestCyl.M_Pump3Add(bAdd:= FALSE)
      //AND THIS^.itfPump3Pressure.M_SetLimit(ePressureType:= E_PRESSURE_TYPE.PERCENT, rLimit:= 0)
			THEN
        THIS^.stSeqCtrlGeneral.iInternalSeqStateCase := 40; 
			END_IF
      
    40: // Disable pump 4
      IF TRUE 
			AND THIS^.itfTestCyl.M_Pump4Add(bAdd:= FALSE)
      //AND THIS^.itfPump4Pressure.M_SetLimit(ePressureType:= E_PRESSURE_TYPE.PERCENT, rLimit:= 0)
			THEN
        THIS^.stSeqCtrlGeneral.iInternalSeqStateCase := 60; 
			END_IF
      
    60: // Move Test Cylinder 1 to HP - Add low pressure circuit to counter cylinder
      IF TRUE 
			AND THIS^.itfCounterCyl.M_LowPressureCircuit(bAdd:= TRUE)
			THEN 
				THIS^.stSeqCtrlGeneral.iInternalSeqStateCase := 70; 
			END_IF
      
    70: // Move Test Cylinder 1 to HP - Move to HP (Min position)
      IF TRUE
      AND THIS^.bDoubleActing
			THEN 
				THIS^.stSeqCtrlGeneral.iInternalSeqStateCase := 71; 
      ELSE
        THIS^.stSeqCtrlGeneral.iInternalSeqStateCase := 72; 
			END_IF
      
    71: // Move Test Cylinder 1 to HP - Move to HP (Min position)
      IF TRUE
      AND THIS^.itfTestCyl.M_ToHP(ePressureType:= E_PRESSURE_TYPE.FORCE, 
                                  rWorkPressure:= THIS^.rWorkForceBTmp * 1000, 
                                  bPressureRegulation:= FALSE,
                                  eSpeedType:= E_SPEED_TYPE.PERCENT, 
                                  rSpeed:= 50)
      AND THIS^.itfCounterCyl.M_ToHP(ePressureType:= E_PRESSURE_TYPE.VALUE, 
                                     rWorkPressure:= 0, 
                                     bPressureRegulation:= FALSE,
                                     eSpeedType:= E_SPEED_TYPE.PERCENT, 
                                     rSpeed:= 50)
			THEN 
        THIS^.stSeqCtrlGeneral.iInternalSeqStateCase := 80;
			END_IF
      
    72: // Move Test Cylinder 1 to HP - Move to HP (Min position)
      IF TRUE
      AND THIS^.itfTestCyl.M_ToHP(ePressureType:= E_PRESSURE_TYPE.VALUE, 
                                  rWorkPressure:= 0, 
                                  bPressureRegulation:= FALSE,
                                  eSpeedType:= E_SPEED_TYPE.PERCENT, 
                                  rSpeed:= 50)
      AND THIS^.itfCounterCyl.M_ToWP(ePressureType:= E_PRESSURE_TYPE.FORCE, 
                                   rWorkPressure:= THIS^.rLoadForceATmp * 1000, 
                                   bPressureRegulation:= FALSE,
                                   eSpeedType:= E_SPEED_TYPE.PERCENT, 
                                   rSpeed:= 50)
			THEN 
        THIS^.stSeqCtrlGeneral.iInternalSeqStateCase := 80;
			END_IF
      
    80:	// Delay timer
      IF TRUE 
      AND _m_Delay(DelayTime:= T#3S)
			THEN 
        THIS^.stSeqCtrlGeneral.iInternalSeqStateCase := 81;
			END_IF
      
    81:	// Wait for HP endpos
      IF TRUE 
			THEN 
        IF TRUE 
        AND ABS(THIS^.itfTestCyl.P_PositionAbs - THIS^.lrLastPos) < 0.5
        THEN
				  THIS^.stSeqCtrlGeneral.iInternalSeqStateCase := 1000;
        ELSE
          THIS^.lrLastPos := THIS^.itfTestCyl.P_PositionAbs;
          THIS^.stSeqCtrlGeneral.iInternalSeqStateCase := 80;
        END_IF
			END_IF
      
    1000: // Exit seq - Disable low pressure circuit
      IF TRUE
      AND _m_Delay(DelayTime:= T#1S)
      AND THIS^.itfCounterCyl.M_LowPressureCircuit(bAdd:= FALSE)
			THEN 
				THIS^.stSeqCtrlGeneral.iInternalSeqStateCase := 1010;
			END_IF  
    
    1010: // Exit seq - Stop
      IF TRUE
      AND _m_Delay(DelayTime:= T#1S) 
      AND THIS^.itfTestCyl.M_StopAndLock()
      AND THIS^.itfCounterCyl.M_Stop()
			THEN 
				THIS^.stSeqCtrlGeneral.iInternalSeqStateCase := 1020;
			END_IF
      
    1020: // Set pressure
      IF TRUE 
			AND THIS^.itfCounterCyl.M_SetWorkPressureZero()
      AND THIS^.itfTestCyl.M_SetWorkPressureZero()
			THEN 
				THIS^.stSeqCtrlGeneral.iInternalSeqStateCase := 9999; 
			END_IF
      
	ELSE
		THIS^.stSeqCtrlGeneral.eActiveSeqState:=E_SEQ_GENERAL.DONE;  
	END_CASE
	THIS^.stSeqCtrlGeneral.strExtraInfo:=concat('Internal state: ', TO_STRING(THIS^.stSeqCtrlGeneral.iInternalSeqStateCase));
E_SEQ_GENERAL.DONE:;
E_SEQ_GENERAL.ERROR:;
E_SEQ_GENERAL.TIME_OUT:; 

IF TRUE
AND THIS^.stSeqCtrlGeneral.bTimeOutActiveQuit 
THEN
  THIS^.stSeqCtrlGeneral.strExtraInfo:= 'Bitte quittieren und erneut testen';
  IF TRUE
  //AND itfOpMode.P_QUIT
  THEN
    THIS^.stSeqCtrlGeneral.eActiveSeqState:=E_SEQ_GENERAL.EXECUTE;
	END_IF
  
END_IF

ELSE
  THIS^.stSeqCtrlGeneral.eActiveSeqState:=E_SEQ_GENERAL.ERROR;
END_CASE
END_METHOD

METHOD PRIVATE _m_Seq_MOVE_TO_SET_POS : E_SEQ_PROCESS
VAR_INPUT
END_VAR
VAR
  ActiveSeq: STRING;
END_VAR
//THIS^._m_GeneralStepSetting(StepType:=E_STEP_STATE_TYPE.INIT,
ActiveSeq := TO_STRING(THIS^.eSeq);

CASE THIS^.stSeqCtrlGeneral.eActiveSeqState OF
E_SEQ_GENERAL.READY:;

	
E_SEQ_GENERAL.EXECUTE:;
	IF TRUE
	AND _m_Delay(T#1S)
	THEN
		THIS^.stSeqCtrlGeneral.eActiveSeqState := E_SEQ_GENERAL.RESET;
	END_IF
  
E_SEQ_GENERAL.RESET:;
	stSeqCtrlGeneral.iInternalSeqStateCase := 0;
	IF TRUE
	THEN
		THIS^.stSeqCtrlGeneral.eActiveSeqState := E_SEQ_GENERAL.BUSY;
	END_IF
  
E_SEQ_GENERAL.BUSY:;
	CASE THIS^.stSeqCtrlGeneral.iInternalSeqStateCase OF
		0:	// Entrance step
      IF TRUE 
			AND _m_Delay(T#2S)
			AND THIS^.itfTestCyl.M_ToSetPos(0,0,0)
			THEN 
				THIS^.stSeqCtrlGeneral.iInternalSeqStateCase := 10; 
			END_IF
      
		10: // Step 10
      IF TRUE 
			AND _m_Delay(T#2S) 
			//AND
			THEN 
				THIS^.stSeqCtrlGeneral.iInternalSeqStateCase := 20; 
			END_IF
      
		20: // Step 20
      IF TRUE 
			AND _m_Delay(T#2S) 
			//AND
			THEN 
				THIS^.stSeqCtrlGeneral.iInternalSeqStateCase := 30; 
			END_IF
      
		30:	// Step 30
      IF TRUE 
			AND _m_Delay(T#2S) 
			//AND
			THEN 
				THIS^.stSeqCtrlGeneral.iInternalSeqStateCase := 1000; 
			END_IF
      
    1000: // Exit step
      IF TRUE
			THEN 
				THIS^.stSeqCtrlGeneral.iInternalSeqStateCase := 9999;
			END_IF
      
	ELSE
		THIS^.stSeqCtrlGeneral.eActiveSeqState := E_SEQ_GENERAL.DONE;  
	END_CASE
	THIS^.stSeqCtrlGeneral.strExtraInfo := CONCAT('Internal state: ', TO_STRING(THIS^.stSeqCtrlGeneral.iInternalSeqStateCase));
E_SEQ_GENERAL.DONE:;
E_SEQ_GENERAL.ERROR:;
E_SEQ_GENERAL.TIME_OUT:; 

IF TRUE
AND THIS^.stSeqCtrlGeneral.bTimeOutActiveQuit 
THEN
  THIS^.stSeqCtrlGeneral.strExtraInfo := 'Bitte quittieren und erneut testen';
  IF TRUE
  //AND itfOpMode.P_QUIT
  THEN
    THIS^.stSeqCtrlGeneral.eActiveSeqState := E_SEQ_GENERAL.EXECUTE;
	END_IF
  
END_IF

ELSE
  THIS^.stSeqCtrlGeneral.eActiveSeqState := E_SEQ_GENERAL.ERROR;
END_CASE
END_METHOD

METHOD PRIVATE _m_Seq_RESET_DISTANCE : BOOL
VAR_INPUT
END_VAR
VAR
  ActiveSeq: STRING;
END_VAR
//THIS^._m_GeneralStepSetting(StepType:=E_STEP_STATE_TYPE.INIT,
ActiveSeq := TO_STRING(THIS^.eSeq);

CASE THIS^.stSeqCtrlGeneral.eActiveSeqState OF
E_SEQ_GENERAL.READY:;
	
E_SEQ_GENERAL.EXECUTE:;
	IF TRUE
	//AND _m_Delay(T#1S)
	THEN
		THIS^.stSeqCtrlGeneral.eActiveSeqState := E_SEQ_GENERAL.RESET;
	END_IF
  
E_SEQ_GENERAL.RESET:;
	stSeqCtrlGeneral.iInternalSeqStateCase := 0;
	IF TRUE
	THEN
		THIS^.stSeqCtrlGeneral.eActiveSeqState := E_SEQ_GENERAL.BUSY;
	END_IF
  
E_SEQ_GENERAL.BUSY:;
	CASE THIS^.stSeqCtrlGeneral.iInternalSeqStateCase OF
		0: // Check if enabled
      IF TRUE 
			THEN 
        THIS^.lrDistanceInM := 0.0;
        THIS^.lrLastRecordPos := 0.0;
        THIS^.uiRecordDelayCycleCount := 0;
        THIS^.stSeqCtrlGeneral.iInternalSeqStateCase := 1000;
			END_IF
      
    1000: // Exit step
      IF TRUE
      AND THIS^.itfCounterCyl.M_LowPressureCircuit(bAdd:= FALSE)
			THEN 
				THIS^.stSeqCtrlGeneral.iInternalSeqStateCase := 9999;
			END_IF
      
	ELSE
		THIS^.stSeqCtrlGeneral.eActiveSeqState:=E_SEQ_GENERAL.DONE;  
	END_CASE
	THIS^.stSeqCtrlGeneral.strExtraInfo:=concat('Internal state: ', TO_STRING(THIS^.stSeqCtrlGeneral.iInternalSeqStateCase));
E_SEQ_GENERAL.DONE:;
E_SEQ_GENERAL.ERROR:;
E_SEQ_GENERAL.TIME_OUT:; 

IF TRUE
AND THIS^.stSeqCtrlGeneral.bTimeOutActiveQuit 
THEN
  THIS^.stSeqCtrlGeneral.strExtraInfo:= 'Bitte quittieren und erneut testen';
  IF TRUE
  //AND itfOpMode.P_QUIT
  THEN
    THIS^.stSeqCtrlGeneral.eActiveSeqState:=E_SEQ_GENERAL.EXECUTE;
	END_IF
  
END_IF

ELSE
  THIS^.stSeqCtrlGeneral.eActiveSeqState:=E_SEQ_GENERAL.ERROR;
END_CASE
END_METHOD

METHOD PRIVATE _m_Seq_STOP : E_SEQ_PROCESS
VAR_INPUT
END_VAR
VAR
  ActiveSeq: STRING;
END_VAR
//THIS^._m_GeneralStepSetting(StepType:=E_STEP_STATE_TYPE.INIT,
ActiveSeq := TO_STRING(THIS^.eSeq);

CASE THIS^.stSeqCtrlGeneral.eActiveSeqState OF
E_SEQ_GENERAL.READY:;

E_SEQ_GENERAL.EXECUTE:;
	IF TRUE
	THEN
		THIS^.stSeqCtrlGeneral.eActiveSeqState := E_SEQ_GENERAL.RESET;
	END_IF
  
E_SEQ_GENERAL.RESET:;
	stSeqCtrlGeneral.iInternalSeqStateCase := 0;
  IF TRUE
	THEN
    THIS^.udiCurrentCycle := 1;
		THIS^.stSeqCtrlGeneral.eActiveSeqState := E_SEQ_GENERAL.BUSY;
	END_IF
  
E_SEQ_GENERAL.BUSY:;
	CASE THIS^.stSeqCtrlGeneral.iInternalSeqStateCase OF
    0: // Set pressure
      IF TRUE 
			AND THIS^.itfCounterCyl.M_SetWorkPressureZero()
      AND THIS^.itfTestCyl.M_SetWorkPressureZero()
			THEN 
				THIS^.stSeqCtrlGeneral.iInternalSeqStateCase := 10; 
			END_IF
      
    10: // Disable low pressure circuit to counter cylinder
      IF TRUE 
			AND THIS^.itfCounterCyl.M_LowPressureCircuit(bAdd:= FALSE)
			THEN 
				THIS^.stSeqCtrlGeneral.iInternalSeqStateCase := 20; 
			END_IF
      
    20: // Vent cylinder - Move to WP (Max position)
      IF TRUE
      AND THIS^.itfTestCyl.M_StopAndLock()
      AND THIS^.itfCounterCyl.M_Stop()
			THEN 
				THIS^.stSeqCtrlGeneral.iInternalSeqStateCase := 30; 
			END_IF
      
    30: // Disable pump 2
      IF TRUE 
			AND THIS^.itfTestCyl.M_Pump2Add(bAdd:= FALSE)
      //AND THIS^.itfPump2Pressure.M_SetLimit(ePressureType:= E_PRESSURE_TYPE.PERCENT, rLimit:= 0)
			THEN
        THIS^.stSeqCtrlGeneral.iInternalSeqStateCase := 40; 
			END_IF
      
    40: // Disable pump 3
      IF TRUE 
			AND THIS^.itfTestCyl.M_Pump3Add(bAdd:= FALSE)
      //AND THIS^.itfPump3Pressure.M_SetLimit(ePressureType:= E_PRESSURE_TYPE.PERCENT, rLimit:= 0)
			THEN
        THIS^.stSeqCtrlGeneral.iInternalSeqStateCase := 50; 
			END_IF
      
    50: // Disable pump 4
      IF TRUE 
			AND THIS^.itfTestCyl.M_Pump4Add(bAdd:= FALSE)
      //AND THIS^.itfPump4Pressure.M_SetLimit(ePressureType:= E_PRESSURE_TYPE.PERCENT, rLimit:= 0)
			THEN
        THIS^.stSeqCtrlGeneral.iInternalSeqStateCase := 1000; 
			END_IF
      
    1000: // Exit step
      IF TRUE
			THEN 
				THIS^.stSeqCtrlGeneral.iInternalSeqStateCase := 9999;
			END_IF
      
	ELSE
		THIS^.stSeqCtrlGeneral.eActiveSeqState:=E_SEQ_GENERAL.DONE;  
	END_CASE
	THIS^.stSeqCtrlGeneral.strExtraInfo:=concat('Internal state: ', TO_STRING(THIS^.stSeqCtrlGeneral.iInternalSeqStateCase));
E_SEQ_GENERAL.DONE:;
E_SEQ_GENERAL.ERROR:;
E_SEQ_GENERAL.TIME_OUT:; 

IF TRUE
AND THIS^.stSeqCtrlGeneral.bTimeOutActiveQuit 
THEN
  THIS^.stSeqCtrlGeneral.strExtraInfo:= 'Bitte quittieren und erneut testen';
  IF TRUE
  //AND itfOpMode.P_QUIT
  THEN
    THIS^.stSeqCtrlGeneral.eActiveSeqState:=E_SEQ_GENERAL.EXECUTE;
	END_IF
  
END_IF

ELSE
  THIS^.stSeqCtrlGeneral.eActiveSeqState:=E_SEQ_GENERAL.ERROR;
END_CASE
END_METHOD

METHOD PRIVATE _m_Seq_STOP_ENGINE : E_SEQ_PROCESS
VAR_INPUT
END_VAR
VAR
	ActiveSeq: STRING;
END_VAR
VAR
	
END_VAR
//THIS^._m_GeneralStepSetting(StepType:=E_STEP_STATE_TYPE.INIT,
ActiveSeq := TO_STRING(THIS^.eSeq);

CASE THIS^.stSeqCtrlGeneral.eActiveSeqState OF
E_SEQ_GENERAL.READY:;

	
E_SEQ_GENERAL.EXECUTE:;
	IF TRUE
	THEN
		THIS^.stSeqCtrlGeneral.eActiveSeqState := E_SEQ_GENERAL.RESET;
	END_IF
E_SEQ_GENERAL.RESET:;
	stSeqCtrlGeneral.iInternalSeqStateCase := 0;
  
	IF TRUE
	THEN
		THIS^.stSeqCtrlGeneral.eActiveSeqState := E_SEQ_GENERAL.BUSY;
	END_IF
E_SEQ_GENERAL.BUSY:;
	CASE THIS^.stSeqCtrlGeneral.iInternalSeqStateCase OF
		0:  // Switch off the counter cylinder pump
      IF TRUE 
			AND THIS^.itfCounterCylPump.M_Off()
			THEN 
				THIS^.stSeqCtrlGeneral.iInternalSeqStateCase := 10; 
			END_IF
      
    10: // Enable bypass
      IF TRUE 
			AND THIS^.itfCounterCylPump.M_Bypass(bEnable:= TRUE)
			THEN 
				THIS^.stSeqCtrlGeneral.iInternalSeqStateCase := 20; 
			END_IF
      
    20: // Switch off the test cylinder pump
      IF TRUE 
			AND THIS^.itfTestCylPump.M_Off()
			THEN 
				THIS^.stSeqCtrlGeneral.iInternalSeqStateCase := 1000; 
			END_IF
      
    1000: // Exit step
      IF TRUE
			THEN 
				THIS^.stSeqCtrlGeneral.iInternalSeqStateCase := 9999;
			END_IF
      
	ELSE
		THIS^.stSeqCtrlGeneral.eActiveSeqState := E_SEQ_GENERAL.DONE;  
	END_CASE
	THIS^.stSeqCtrlGeneral.strExtraInfo := CONCAT('Internal state: ', TO_STRING(THIS^.stSeqCtrlGeneral.iInternalSeqStateCase));
E_SEQ_GENERAL.DONE:;
E_SEQ_GENERAL.ERROR:;
E_SEQ_GENERAL.TIME_OUT:; 

IF TRUE
AND THIS^.stSeqCtrlGeneral.bTimeOutActiveQuit 
THEN
  THIS^.stSeqCtrlGeneral.strExtraInfo := 'Bitte quittieren und erneut testen';
  IF TRUE
  //AND itfOpMode.P_QUIT
  THEN
    THIS^.stSeqCtrlGeneral.eActiveSeqState := E_SEQ_GENERAL.EXECUTE;
	END_IF
  
END_IF

ELSE
  THIS^.stSeqCtrlGeneral.eActiveSeqState := E_SEQ_GENERAL.ERROR;
END_CASE
END_METHOD

METHOD PRIVATE _m_Seq_VENT_CYLINDER : E_SEQ_PROCESS
VAR_INPUT
END_VAR
VAR
  ActiveSeq: STRING;
END_VAR
//THIS^._m_GeneralStepSetting(StepType:=E_STEP_STATE_TYPE.INIT,
ActiveSeq := TO_STRING(THIS^.eSeq);

// Distance record
_m_DistanceRecord();

CASE THIS^.stSeqCtrlGeneral.eActiveSeqState OF
E_SEQ_GENERAL.READY:;

E_SEQ_GENERAL.EXECUTE:;
	IF TRUE
	AND _m_Delay(T#1S)
	THEN
		THIS^.stSeqCtrlGeneral.eActiveSeqState := E_SEQ_GENERAL.RESET;
	END_IF
  
E_SEQ_GENERAL.RESET:;
	stSeqCtrlGeneral.iInternalSeqStateCase := 0;
  IF TRUE
	THEN
    THIS^.udiCurrentCycle := 1;
		THIS^.stSeqCtrlGeneral.eActiveSeqState := E_SEQ_GENERAL.BUSY;
	END_IF
  
E_SEQ_GENERAL.BUSY:;
	CASE THIS^.stSeqCtrlGeneral.iInternalSeqStateCase OF
    0: // Check if enable
      IF TRUE
      AND THIS^.bEnable 
      THEN
        THIS^.stSeqCtrlGeneral.iInternalSeqStateCase := 10; 
      ELSE
        THIS^.stSeqCtrlGeneral.iInternalSeqStateCase := 9999; 
			END_IF

    10: // Disable low pressure mode
      IF TRUE 
      AND _m_Delay(DelayTime:= T#3S)
			AND THIS^.itfTestCyl.M_LowPressureMode(bSet:= FALSE, ePressureType:= E_PRESSURE_TYPE.VALUE, rWorkPressure:= 0)
			THEN 
				THIS^.stSeqCtrlGeneral.iInternalSeqStateCase := 20; 
			END_IF
      
    20: // Disable pump 2
      IF TRUE 
			AND THIS^.itfTestCyl.M_Pump2Add(bAdd:= FALSE)
      //AND THIS^.itfPump2Pressure.M_SetLimit(ePressureType:= E_PRESSURE_TYPE.PERCENT, rLimit:= 0)
			THEN
        THIS^.stSeqCtrlGeneral.iInternalSeqStateCase := 30; 
			END_IF
      
    30: // Disable pump 3
      IF TRUE 
			AND THIS^.itfTestCyl.M_Pump3Add(bAdd:= FALSE)
      //AND THIS^.itfPump3Pressure.M_SetLimit(ePressureType:= E_PRESSURE_TYPE.PERCENT, rLimit:= 0)
			THEN
        THIS^.stSeqCtrlGeneral.iInternalSeqStateCase := 40; 
			END_IF
      
    40: // Disable pump 4
      IF TRUE 
			AND THIS^.itfTestCyl.M_Pump4Add(bAdd:= FALSE)
      //AND THIS^.itfPump4Pressure.M_SetLimit(ePressureType:= E_PRESSURE_TYPE.PERCENT, rLimit:= 0)
			THEN
        THIS^.stSeqCtrlGeneral.iInternalSeqStateCase := 50; 
			END_IF
      
    50: // Vent cylinder - Choice step
      IF TRUE 
			THEN 
        IF THIS^.udiCurrentCycle > THIS^.uiVentCount THEN
          THIS^.stSeqCtrlGeneral.iInternalSeqStateCase := 1000; 
        ELSE
          THIS^.stSeqCtrlGeneral.iInternalSeqStateCase := 60; 
				END_IF
			END_IF
      
    60: // Vent cylinder - Add low pressure circuit to counter cylinder
      IF TRUE 
			AND THIS^.itfCounterCyl.M_LowPressureCircuit(bAdd:= TRUE)
			THEN 
				THIS^.stSeqCtrlGeneral.iInternalSeqStateCase := 70; 
			END_IF
      
    70: // Vent cylinder - Move to WP (Max position)
      IF TRUE
      AND NOT THIS^.bCylinderDecoupled
			THEN 
				THIS^.stSeqCtrlGeneral.iInternalSeqStateCase := 71; 
      ELSE
        THIS^.stSeqCtrlGeneral.iInternalSeqStateCase := 72; 
			END_IF
      
    71: // Vent cylinder - Move to WP (Max position)
      IF TRUE
      AND THIS^.itfTestCyl.M_ToWP(ePressureType:= E_PRESSURE_TYPE.FORCE, 
                                  rWorkPressure:= THIS^.rWorkForceATmp * 1000, 
                                  bPressureRegulation:= FALSE,
                                  eSpeedType:= E_SPEED_TYPE.PERCENT, 
                                  rSpeed:= 50)
      AND THIS^.itfCounterCyl.M_ToWP(ePressureType:= E_PRESSURE_TYPE.VALUE, 
                                     rWorkPressure:= 0,
                                     bPressureRegulation:= FALSE, 
                                     eSpeedType:= E_SPEED_TYPE.PERCENT, 
                                     rSpeed:= 50)
			THEN 
				THIS^.stSeqCtrlGeneral.iInternalSeqStateCase := 80; 
			END_IF
      
    72: // Vent cylinder - Move to WP (Max position)
      IF TRUE
      AND THIS^.itfTestCyl.M_ToWP(ePressureType:= E_PRESSURE_TYPE.FORCE, 
                                  rWorkPressure:= THIS^.rWorkForceATmp * 1000, 
                                  bPressureRegulation:= FALSE,
                                  eSpeedType:= E_SPEED_TYPE.PERCENT, 
                                  rSpeed:= 50)
      AND THIS^.itfCounterCyl.M_ToHP(ePressureType:= E_PRESSURE_TYPE.FORCE, 
                                     rWorkPressure:= THIS^.rLoadForceBTmp * 1000,
                                     bPressureRegulation:= FALSE, 
                                     eSpeedType:= E_SPEED_TYPE.PERCENT, 
                                     rSpeed:= 50)
			THEN 
				THIS^.stSeqCtrlGeneral.iInternalSeqStateCase := 80; 
			END_IF
      
    80:	// Delay timer
      IF TRUE 
      AND _m_Delay(DelayTime:= T#3S)
			THEN 
        THIS^.stSeqCtrlGeneral.iInternalSeqStateCase := 81;
			END_IF
      
    81:	// Wait for WP endpos
      IF TRUE 
			THEN 
        IF TRUE 
        AND ABS(THIS^.itfTestCyl.P_PositionAbs - THIS^.lrLastPos) < 0.5
        THEN
          THIS^.stSeqCtrlGeneral.iInternalSeqStateCase := 90;
        ELSE
          THIS^.lrLastPos := THIS^.itfTestCyl.P_PositionAbs;
          THIS^.stSeqCtrlGeneral.iInternalSeqStateCase := 80;
        END_IF
			END_IF
      
    90: // Vent cylinder - Move to HP (Min position)
      IF TRUE
      AND THIS^.bDoubleActing
			THEN 
				THIS^.stSeqCtrlGeneral.iInternalSeqStateCase := 91; 
      ELSE
        THIS^.stSeqCtrlGeneral.iInternalSeqStateCase := 92; 
			END_IF
      
    91: // Vent cylinder - Move to HP (Min position)
      IF TRUE
      AND THIS^.itfTestCyl.M_ToHP(ePressureType:= E_PRESSURE_TYPE.FORCE, 
                                  rWorkPressure:= THIS^.rWorkForceBTmp * 1000, 
                                  bPressureRegulation:= FALSE,
                                  eSpeedType:= E_SPEED_TYPE.PERCENT, 
                                  rSpeed:= 50)
      AND THIS^.itfCounterCyl.M_ToHP(ePressureType:= E_PRESSURE_TYPE.VALUE, 
                                     rWorkPressure:= 0, 
                                     bPressureRegulation:= FALSE,
                                     eSpeedType:= E_SPEED_TYPE.PERCENT, 
                                     rSpeed:= 50)
			THEN 
        THIS^.stSeqCtrlGeneral.iInternalSeqStateCase := 100;
			END_IF
      
    92: // Vent cylinder - Move to HP (Min position)
      IF TRUE
      AND THIS^.itfTestCyl.M_ToHP(ePressureType:= E_PRESSURE_TYPE.VALUE, 
                                  rWorkPressure:= 0, 
                                  bPressureRegulation:= FALSE,
                                  eSpeedType:= E_SPEED_TYPE.PERCENT, 
                                  rSpeed:= 50)
			THEN 
        THIS^.stSeqCtrlGeneral.iInternalSeqStateCase := 93;
			END_IF
      
    93: // Vent cylinder - Move to HP (Min position) - Check if Cylinder decoupled
      IF TRUE
      AND NOT THIS^.bCylinderDecoupled
      THEN
        IF THIS^.itfCounterCyl.M_ToWP(ePressureType:= E_PRESSURE_TYPE.FORCE, 
                                     rWorkPressure:= THIS^.rLoadForceATmp * 1000, 
                                     bPressureRegulation:= FALSE,
                                     eSpeedType:= E_SPEED_TYPE.PERCENT, 
                                     rSpeed:= 50)
			  THEN 
          THIS^.stSeqCtrlGeneral.iInternalSeqStateCase := 100;
        END_IF
      ELSE
        THIS^.stSeqCtrlGeneral.iInternalSeqStateCase := 100;
			END_IF
      
    100:	// Delay timer
      IF TRUE 
      AND _m_Delay(DelayTime:= T#3S)
			THEN 
        THIS^.stSeqCtrlGeneral.iInternalSeqStateCase := 101;
			END_IF
      
    101:	// Wait for HP endpos
      IF TRUE 
			THEN 
        IF TRUE 
        AND ABS(THIS^.itfTestCyl.P_PositionAbs - THIS^.lrLastPos) < 0.5
        THEN
          THIS^.udiCurrentCycle := THIS^.udiCurrentCycle + 1;
				  THIS^.stSeqCtrlGeneral.iInternalSeqStateCase := 50; // Jump back
        ELSE
          THIS^.lrLastPos := THIS^.itfTestCyl.P_PositionAbs;
          THIS^.stSeqCtrlGeneral.iInternalSeqStateCase := 100;
        END_IF
			END_IF
      
    1000: // Exit seq - Disable low pressure circuit
      IF TRUE
      AND _m_Delay(DelayTime:= T#1S)
      AND THIS^.itfCounterCyl.M_LowPressureCircuit(bAdd:= FALSE)
			THEN 
				THIS^.stSeqCtrlGeneral.iInternalSeqStateCase := 1010;
			END_IF  
    
    1010: // Exit seq - Stop
      IF TRUE
      AND _m_Delay(DelayTime:= T#1S) 
      AND THIS^.itfTestCyl.M_StopAndLock()
      AND THIS^.itfCounterCyl.M_Stop()
			THEN 
				THIS^.stSeqCtrlGeneral.iInternalSeqStateCase := 1020;
			END_IF
      
    1020: // Set pressure
      IF TRUE 
			AND THIS^.itfCounterCyl.M_SetWorkPressureZero()
      AND THIS^.itfTestCyl.M_SetWorkPressureZero()
			THEN 
				THIS^.stSeqCtrlGeneral.iInternalSeqStateCase := 9999; 
			END_IF
      
	ELSE
		THIS^.stSeqCtrlGeneral.eActiveSeqState:=E_SEQ_GENERAL.DONE;  
	END_CASE
	THIS^.stSeqCtrlGeneral.strExtraInfo:=concat('Internal state: ', TO_STRING(THIS^.stSeqCtrlGeneral.iInternalSeqStateCase));
E_SEQ_GENERAL.DONE:;
E_SEQ_GENERAL.ERROR:;
E_SEQ_GENERAL.TIME_OUT:; 

IF TRUE
AND THIS^.stSeqCtrlGeneral.bTimeOutActiveQuit 
THEN
  THIS^.stSeqCtrlGeneral.strExtraInfo:= 'Bitte quittieren und erneut testen';
  IF TRUE
  //AND itfOpMode.P_QUIT
  THEN
    THIS^.stSeqCtrlGeneral.eActiveSeqState:=E_SEQ_GENERAL.EXECUTE;
	END_IF
  
END_IF

ELSE
  THIS^.stSeqCtrlGeneral.eActiveSeqState:=E_SEQ_GENERAL.ERROR;
END_CASE
END_METHOD

METHOD PRIVATE _m_SequenceManager
VAR_INPUT
END_VAR
IF FALSE
//AND THIS^.eActiveSeqState=DONE 
AND eLastSeq<>eSeq
THEN
	IF THIS^.stSeqCtrlGeneral.eActiveSeqState<>E_SEQ_GENERAL.EXECUTE THEN
		THIS^.stSeqCtrlGeneral.eActiveSeqState:=E_SEQ_GENERAL.READY;
	END_IF
END_IF

eSeq := eNextSeq;

//DelayTimer und TimeOut Timer verwalten
stSeqCtrlGeneral.bActiveStep := TRUE
				                        AND eLastSeq = eSeq
				                        AND stSeqCtrlGeneral.eLastActiveSeqState = stSeqCtrlGeneral.eActiveSeqState
				                        AND	stSeqCtrlGeneral.iLastInternalSeqStateCase = stSeqCtrlGeneral.iInternalSeqStateCase;
			
IF NOT stSeqCtrlGeneral.bActiveStep THEN
	stSeqCtrlGeneral.bDelayActive:=FALSE;
	stSeqCtrlGeneral.bTimeOutActiveQuit:=FALSE;
	stSeqCtrlGeneral.bTimeOutActiveNoQuit:=FALSE;
  THIS^.stSeqCtrlGeneral.strExtraInfo:='';
END_IF

_m_SaveLastStep();
stSeqCtrlGeneral.tonDelay	(IN:=stSeqCtrlGeneral.bActiveStep AND stSeqCtrlGeneral.bDelayActive, 		PT:=stSeqCtrlGeneral.tDelay);
stSeqCtrlGeneral.tonTimeOut	(IN:=stSeqCtrlGeneral.bActiveStep AND (stSeqCtrlGeneral.bTimeOutActiveNoQuit OR stSeqCtrlGeneral.bTimeOutActiveQuit), 	PT:=stSeqCtrlGeneral.tTimeOut);
stSeqCtrlGeneral.tonStepTime	(IN:= stSeqCtrlGeneral.bActiveStep, PT:= T#24H);

IF stSeqCtrlGeneral.tonTimeOut.Q  THEN
	stSeqCtrlGeneral.eActiveSeqState:=E_SEQ_GENERAL.TIME_OUT;
END_IF

IF stSeqCtrlGeneral.iError<>0 THEN
	eSeq:=E_SEQ_PROCESS.ERROR_SEQ;
END_IF



eLastSeq					:=	eSeq;
stSeqCtrlGeneral.eLastActiveSeqState			:=	stSeqCtrlGeneral.eActiveSeqState;
stSeqCtrlGeneral.iLastInternalSeqStateCase	:=	stSeqCtrlGeneral.iInternalSeqStateCase;

// Reset set ready state
IF THIS^.stSeqCtrlGeneral.bExitSetReadyState THEN
  THIS^.stSeqCtrlGeneral.bExitSetReadyState := FALSE;
END_IF
END_METHOD

METHOD PRIVATE _m_TimeOut : BOOL
VAR_INPUT
	bTimeoutActiveToQuit:	BOOL;
	bTimeOutActiveNoQuit:	BOOL;
	tTimeOut:				TIME;	
END_VAR
THIS^.stSeqCtrlGeneral.bTimeOutActiveQuit:=	bTimeoutActiveToQuit;
THIS^.stSeqCtrlGeneral.bTimeOutActiveNoQuit:=	bTimeOutActiveNoQuit;
THIS^.stSeqCtrlGeneral.tTimeOut:=			tTimeOut;
_m_TimeOut:=FALSE;
IF THIS^.stSeqCtrlGeneral.tonTimeOut.Q THEN
	_m_TimeOut:=TRUE;
END_IF
END_METHOD

METHOD FB_init : BOOL
VAR_INPUT
	bInitRetains : BOOL; // if TRUE, the retain variables are initialized (warm start / cold start)
	bInCopyCode : BOOL;  // if TRUE, the instance afterwards gets moved into the copy code (online change)
  
  itfOpMode:											                        I_OP_MODE;
  itfEventLogger:                                         I_EVENT_LOGGER; 
  itfTimer:                                               I_CLOCK; 
  itfCounterCyl:                                          I_CYLINDER_DA_COUNTER;
  itfTestCyl:                                             I_CYLINDER_DA_TESTDEV1;
  itfCounterCylPump:                                      I_PUMP_WITH_BYPASS;
  itfTestCylPump:                                         I_PUMP;
  itfPump2Pressure:                                       I_PRV_PROP;
  itfPump3Pressure:                                       I_PRV_PROP;
  itfPump4Pressure:                                       I_PRV_PROP;
END_VAR
THIS^.itfOpMode := itfOpMode;
THIS^.itfEventLogger := itfEventLogger;
THIS^.itfTimer := itfTimer;
THIS^.itfCounterCyl := itfCounterCyl;
THIS^.itfTestCyl := itfTestCyl;
THIS^.itfCounterCylPump := itfCounterCylPump;
THIS^.itfTestCylPump := itfTestCylPump;
THIS^.itfPump2Pressure := itfPump2Pressure;
THIS^.itfPump3Pressure := itfPump3Pressure;
THIS^.itfPump4Pressure := itfPump4Pressure;
END_METHOD

METHOD M_BreakPressureDet : BOOL
VAR_INPUT
  stBreakPressureParams:                ST_RECIPE_BREAK_PRESSURE;
END_VAR
M_BreakPressureDet := THIS^.stSeqCtrlGeneral.eActiveSeqState = E_SEQ_GENERAL.DONE;

// Assign input
THIS^.stBPDParams := stBreakPressureParams;

IF THIS^.stSeqCtrlGeneral.eActiveSeqState = E_SEQ_GENERAL.READY THEN
  THIS^.eNextSeq := E_SEQ_PROCESS.BREAK_PRESSURE_DET;
  THIS^.stSeqCtrlGeneral.eActiveSeqState := E_SEQ_GENERAL.EXECUTE;
END_IF
END_METHOD

METHOD M_EnduranceRun : BOOL
VAR_INPUT
  udiCycles:                            UDINT;
  stEnduranceRunParams:                 ST_RECIPE_ENDURANCE_RUN;
END_VAR
M_EnduranceRun := THIS^.stSeqCtrlGeneral.eActiveSeqState = E_SEQ_GENERAL.DONE;

// Assign input
THIS^.udiERCycles := udiCycles;
THIS^.stERParams := stEnduranceRunParams;

// General
IF THIS^.stSeqCtrlGeneral.eActiveSeqState = E_SEQ_GENERAL.READY THEN
  THIS^.eNextSeq := E_SEQ_PROCESS.ENDURANCE_RUN;
  THIS^.stSeqCtrlGeneral.eActiveSeqState := E_SEQ_GENERAL.EXECUTE;
END_IF
END_METHOD

METHOD M_LeakTest1 : BOOL
VAR_INPUT
  stLeakTest1Params:                 ST_RECIPE_LEAK_TEST1;
END_VAR
M_LeakTest1 := THIS^.stSeqCtrlGeneral.eActiveSeqState = E_SEQ_GENERAL.DONE;

// Assign input
THIS^.stLT1Params := stLeakTest1Params;

// General
IF THIS^.stSeqCtrlGeneral.eActiveSeqState = E_SEQ_GENERAL.READY THEN
  THIS^.eNextSeq := E_SEQ_PROCESS.LEAK_TEST_1;
  THIS^.stSeqCtrlGeneral.eActiveSeqState := E_SEQ_GENERAL.EXECUTE;
END_IF
END_METHOD

METHOD M_LeakTest2 : BOOL
VAR_INPUT
  stLeakTest2Params:                 ST_RECIPE_LEAK_TEST2;
END_VAR
M_LeakTest2 := THIS^.stSeqCtrlGeneral.eActiveSeqState = E_SEQ_GENERAL.DONE;

// Assign input
THIS^.stLT2Params := stLeakTest2Params;

// General
IF THIS^.stSeqCtrlGeneral.eActiveSeqState = E_SEQ_GENERAL.READY THEN
  THIS^.eNextSeq := E_SEQ_PROCESS.LEAK_TEST_2;
  THIS^.stSeqCtrlGeneral.eActiveSeqState := E_SEQ_GENERAL.EXECUTE;
END_IF
END_METHOD

METHOD M_MaxSpeedRecord : BOOL
VAR_INPUT 
  stEnduranceRunParams:                 ST_RECIPE_ENDURANCE_RUN;
END_VAR
M_MaxSpeedRecord := THIS^.stSeqCtrlGeneral.eActiveSeqState = E_SEQ_GENERAL.DONE;

// Assign input
THIS^.stERParams := stEnduranceRunParams;

// General
IF THIS^.stSeqCtrlGeneral.eActiveSeqState = E_SEQ_GENERAL.READY THEN
  THIS^.eNextSeq := E_SEQ_PROCESS.MAX_SPEED_RECORD;
  THIS^.stSeqCtrlGeneral.eActiveSeqState := E_SEQ_GENERAL.EXECUTE;
END_IF
END_METHOD

METHOD M_MeasureStrokeLength : BOOL
VAR_INPUT
  bCylinderDecoupled:             BOOL;
  rWorkForceA:                    REAL;
  rWorkForceB:                    REAL;
  rLoadForceA:                    REAL;
  rLoadForceB:                    REAL;
END_VAR
M_MeasureStrokeLength := THIS^.stSeqCtrlGeneral.eActiveSeqState = E_SEQ_GENERAL.DONE;

// Assign input
THIS^.bCylinderDecoupled := bCylinderDecoupled;
THIS^.rWorkForceATmp := rWorkForceA;
THIS^.rWorkForceBTmp := rWorkForceB;
THIS^.rLoadForceATmp := rLoadForceA;
THIS^.rLoadForceBTmp := rLoadForceB;

IF THIS^.stSeqCtrlGeneral.eActiveSeqState = E_SEQ_GENERAL.READY THEN
  THIS^.eNextSeq := E_SEQ_PROCESS.MEASURE_STROKE_LENGTH;
  THIS^.stSeqCtrlGeneral.eActiveSeqState := E_SEQ_GENERAL.EXECUTE;
END_IF
END_METHOD

METHOD M_MoveTestCyl1ToHP : BOOL
VAR_INPUT
  rWorkForceA:                    REAL;
  rWorkForceB:                    REAL;
  rLoadForceA:                    REAL;
  rLoadForceB:                    REAL;
END_VAR
M_MoveTestCyl1ToHP := THIS^.stSeqCtrlGeneral.eActiveSeqState = E_SEQ_GENERAL.DONE;

// Assign input
THIS^.rWorkForceATmp := rWorkForceA;
THIS^.rWorkForceBTmp := rWorkForceB;
THIS^.rLoadForceATmp := rLoadForceA;
THIS^.rLoadForceBTmp := rLoadForceB;

IF THIS^.stSeqCtrlGeneral.eActiveSeqState = E_SEQ_GENERAL.READY THEN
  THIS^.eNextSeq := E_SEQ_PROCESS.MOVE_CYL_TO_HP;
  THIS^.stSeqCtrlGeneral.eActiveSeqState := E_SEQ_GENERAL.EXECUTE;
END_IF
END_METHOD

METHOD M_MoveToSetPos : BOOL
M_MoveToSetPos := THIS^.stSeqCtrlGeneral.eActiveSeqState = E_SEQ_GENERAL.DONE;

IF THIS^.stSeqCtrlGeneral.eActiveSeqState = E_SEQ_GENERAL.READY THEN
  THIS^.eNextSeq := E_SEQ_PROCESS.MOVE_TO_SET_POS;
  THIS^.stSeqCtrlGeneral.eActiveSeqState := E_SEQ_GENERAL.EXECUTE;
END_IF
END_METHOD

METHOD M_Reset : BOOL
M_Reset := THIS^.stSeqCtrlGeneral.eActiveSeqState = E_SEQ_GENERAL.DONE;

IF THIS^.stSeqCtrlGeneral.eActiveSeqState = E_SEQ_GENERAL.READY THEN
  THIS^.eNextSeq := E_SEQ_PROCESS.INIT;
  THIS^.stSeqCtrlGeneral.eActiveSeqState := E_SEQ_GENERAL.EXECUTE;
END_IF
END_METHOD

METHOD M_ResetDistance : BOOL
M_ResetDistance := THIS^.stSeqCtrlGeneral.eActiveSeqState = E_SEQ_GENERAL.DONE;

// General
IF stSeqCtrlGeneral.eActiveSeqState = E_SEQ_GENERAL.READY THEN
  THIS^.eNextSeq := E_SEQ_PROCESS.RESET_DISTANCE;
  stSeqCtrlGeneral.eActiveSeqState := E_SEQ_GENERAL.EXECUTE;
END_IF
END_METHOD

{warning 'Methodenimplementierung hinzufügen'}
(*=== Method: M_Run  ============================================

 @brief: Here is the global code (Timer, Event, Flange,...)*)
METHOD M_Run
END_METHOD

METHOD M_SetEnableState : BOOL
VAR_INPUT
	bEnable:        BOOL;
END_VAR
THIS^.bEnable := bEnable;
END_METHOD

METHOD M_SetReady : BOOL
VAR_INPUT
END_VAR
M_SetReady := TRUE
              AND THIS^.stSeqCtrlGeneral.eActiveSeqState = E_SEQ_GENERAL.READY
              AND THIS^.eSeq = E_SEQ_PROCESS.BASE;

THIS^.stSeqCtrlGeneral.eActiveSeqState := E_SEQ_GENERAL.READY;
THIS^.eNextSeq := E_SEQ_PROCESS.BASE;
END_METHOD

METHOD M_Stop : BOOL
M_Stop := THIS^.stSeqCtrlGeneral.eActiveSeqState = E_SEQ_GENERAL.DONE;

IF THIS^.stSeqCtrlGeneral.eActiveSeqState = E_SEQ_GENERAL.READY THEN
  THIS^.eNextSeq := E_SEQ_PROCESS.STOP;
  THIS^.stSeqCtrlGeneral.eActiveSeqState := E_SEQ_GENERAL.EXECUTE;
END_IF
END_METHOD

METHOD M_StopEngine : BOOL
M_StopEngine := THIS^.stSeqCtrlGeneral.eActiveSeqState = E_SEQ_GENERAL.DONE;

IF THIS^.stSeqCtrlGeneral.eActiveSeqState = E_SEQ_GENERAL.READY THEN
  THIS^.eNextSeq := E_SEQ_PROCESS.STOP_ENGINE;
  THIS^.stSeqCtrlGeneral.eActiveSeqState := E_SEQ_GENERAL.EXECUTE;
END_IF
END_METHOD

METHOD M_VentCylinder : BOOL
VAR_INPUT
  bCylinderDecoupled:             BOOL;
  uiVentCount:                    UINT;
  rWorkForceA:                    REAL;
  rWorkForceB:                    REAL;
  rLoadForceA:                    REAL;
  rLoadForceB:                    REAL;
END_VAR
M_VentCylinder := THIS^.stSeqCtrlGeneral.eActiveSeqState = E_SEQ_GENERAL.DONE;

// Assign input
THIS^.bCylinderDecoupled := bCylinderDecoupled;
THIS^.uiVentCount := uiVentCount;
THIS^.rWorkForceATmp := rWorkForceA;
THIS^.rWorkForceBTmp := rWorkForceB;
THIS^.rLoadForceATmp := rLoadForceA;
THIS^.rLoadForceBTmp := rLoadForceB;

// General
IF THIS^.stSeqCtrlGeneral.eActiveSeqState = E_SEQ_GENERAL.READY THEN
  THIS^.eNextSeq := E_SEQ_PROCESS.VENT_CYLINDER;
  THIS^.stSeqCtrlGeneral.eActiveSeqState := E_SEQ_GENERAL.EXECUTE;
END_IF
END_METHOD

{warning 'Eigenschaftenimplementierung hinzufügen'}
PROPERTY P_CurrentCycle : UDINT
GET
P_CurrentCycle := THIS^.udiCurrentCycle;
END_GET
END_PROPERTY

{warning 'Eigenschaftenimplementierung hinzufügen'}
PROPERTY P_EnableState : BOOL
GET
P_EnableState := THIS^.bEnable;
END_GET
END_PROPERTY

{warning 'Eigenschaftenimplementierung hinzufügen'}
(*=== Property: P_Event  ============================================

 @param [set]: 	Set the Structure "ST_EVENT" from another Object
 @param [get]: 	Return the Structure "ST_EVENT", it contains the actual 
					event of the Object *)
PROPERTY P_Event : GenLib.ST_EVENT
GET
END_GET
SET
END_SET
END_PROPERTY

{warning 'Eigenschaftenimplementierung hinzufügen'}
(*=== Property: P_FullObjectPath  ============================================

 @param [set]: 	Set the Object Path (Clear String of Object)
 @param [get]: 	Return the Objectpath *)
PROPERTY P_FullObjectPath : STRING
GET
END_GET
SET
END_SET
END_PROPERTY

{warning 'Eigenschaftenimplementierung hinzufügen'}
(*=== Property: P_Global_Ack  ============================================

 @param [set]: 	Set the Bit for Ack from another Object
 @param [get]: 	Return the state of Ack Bit*)
PROPERTY P_Global_Ack : BOOL
GET
END_GET
SET
END_SET
END_PROPERTY

{warning 'Eigenschaftenimplementierung hinzufügen'}
(*=== Property: P_GlobalID  ============================================

 @param [set]: 	-
 @param [get]: 	Return the string of instance path*)
PROPERTY P_GlobalID : STRING
GET
END_GET
END_PROPERTY

{warning 'Eigenschaftenimplementierung hinzufügen'}
PROPERTY P_MaxSpeedInMmPerSHP : REAL
GET
P_MaxSpeedInMmPerSHP := THIS^.rMaxSpeedInMmPerSHP;
END_GET
END_PROPERTY

{warning 'Eigenschaftenimplementierung hinzufügen'}
PROPERTY P_MaxSpeedInMmPerSWP : REAL
GET
P_MaxSpeedInMmPerSWP := THIS^.rMaxSpeedInMmPerSWP;
END_GET
END_PROPERTY

{warning 'Eigenschaftenimplementierung hinzufügen'}
PROPERTY P_NokDifference : REAL
GET
P_NokDifference := THIS^.rCurrentNokDifference;
END_GET
END_PROPERTY

{warning 'Eigenschaftenimplementierung hinzufügen'}
PROPERTY P_NokLimitInPercent : UINT
GET
P_NokLimitInPercent := THIS^.uiCurrentNokLimitInPercent;
END_GET
END_PROPERTY

{warning 'Eigenschaftenimplementierung hinzufügen'}
PROPERTY P_ReadyState : BOOL
GET
P_ReadyState := THIS^.stSeqCtrlGeneral.eActiveSeqState = E_SEQ_GENERAL.READY;
END_GET
END_PROPERTY

{warning 'Eigenschaftenimplementierung hinzufügen'}
PROPERTY P_SerialNr : STRING
GET
P_SerialNr := THIS^.strSerialNr;
END_GET
SET
THIS^.strSerialNr := P_SerialNr;
END_SET
END_PROPERTY

{warning 'Eigenschaftenimplementierung hinzufügen'}
PROPERTY P_SpeedEfficiencyFactor : REAL
GET
P_SpeedEfficiencyFactor := THIS^.rSpeedEfficiencyFactor;
END_GET
END_PROPERTY

{warning 'Eigenschaftenimplementierung hinzufügen'}
PROPERTY P_Timer : STRING
GET
P_Timer := THIS^.sTimer;
END_GET
END_PROPERTY

END_FUNCTION_BLOCK

// ---- FUNCTIONS/FUNCTIONS/MATH/F_RoundREAL.TcPOU
FUNCTION F_RoundREAL : REAL
VAR_INPUT
	rValue:					REAL;
	uiDezimalPlace:	UINT;
END_VAR
VAR
	rResult:				REAL;
	uiMultiplier:		UINT := 1;
	i:							UINT;
END_VAR

FOR i := 1 TO uiDezimalPlace BY 1 DO
	uiMultiplier := uiMultiplier * 10;
END_FOR

rResult := TO_REAL(TO_DINT(rValue * uiMultiplier)) / uiMultiplier;

F_RoundREAL := rResult;

END_FUNCTION

// ---- SUBSTATION/STATION_NEST/POU/FB_SEQ_PROCESS_NEST2_4.TcPOU
FUNCTION_BLOCK FB_SEQ_PROCESS_NEST2_4 IMPLEMENTS I_PROCESS_NEST2_4
VAR_INPUT
  bDoubleActing:                                          BOOL := TRUE;
  rMaxSpeedInMmPerSHP:                                    REAL;
  rMaxSpeedInMmPerSWP:                                    REAL;
  rSpeedEfficiencyFactor:                                 REAL;
  uiRecordDelay:                                          UINT;
END_VAR
VAR //General
	{attribute 'instance-path'} 
  {attribute 'noinit'} 
	strInstancePath:									                      STRING;
	bInit: 												                          BOOL:=TRUE;
	strFullObjectPath: 								                      STRING;
	stEvent:											                          ST_EVENT;
	bAck:												                            BOOL;
	bEnable:                                                BOOL;
END_VAR
VAR   // From FB_init	
	itfOpMode:											                        I_OP_MODE; 
  itfEventLogger:                                         I_EVENT_LOGGER; 
  itfTimer:                                               I_CLOCK; 
  itfCounterCyl:                                          I_CYLINDER_DA_COUNTER;
  itfTestCyl:                                             I_CYLINDER_DA_TESTDEV2_4;
  itfCounterCylPump:                                      I_PUMP_WITH_BYPASS;
  itfTestCylPump:                                         I_PUMP;
END_VAR                                      				
VAR	// Step chain control                				
  eSeq, eLastSeq, eNextSeq:					                      E_SEQ_PROCESS; 
  uiSnippetSeq, uiLastSnippetSeq:                         UINT := 0;
                  				
  //eActiveSeqState, eLastActiveSeqState:                 E_SEQ_GENERAL;
	(*
  iInternalSeqStateCase, iLastInternalSeqStateCase:       INT:=0;       
	tonDelay, tonTimeOut, tonStepTime:						          TON;
	tDelay:													                        TIME := T#100MS;
	tTimeOut:												                        TIME := T#100MS;
	tTimeOutExt:											                      TIME := T#100MS;
	bDelayActive, bTimeOutActiveQuit, bTimeOutActiveNoQuit:	BOOL;//Timer Option
	bActiveStep, bDebugAcitve, bDebugNext:					        BOOL;//Debug Option
	i:														                          INT;
 	iError:													                        INT; //ERROR-CODE                    	                   		
	listLastSteps:											                    ARRAY[0..49] OF ST_LAST_STEPS;	
	strExtraInfo:											                      STRING; 
	eStep_Type:												                      E_STEP_STATE_TYPE; 
	bDebugModeActive:										                    BOOL;   
	bWaitForBreakpoint:										                  BOOL;
	bBreakpointActive:										                  BOOL;
	bDebugResume:											                      BOOL;   
	listBreakpoint:											                    ARRAY[0..10] OF  INT;    
*)
i:														                            INT;
stSeqCtrlGeneral:											                    ST_SEQ_CTRL_GEN;     	
END_VAR                                             		
VAR                                                 		
	bMethodeFromExtStarted:									                BOOL;
	bMethodeFromExtActive:									                BOOL;
	bMethodeFromExtDone:									                  BOOL;
	strTemp:												                        STRING;
END_VAR   
VAR
  strSerialNr:                                            STRING;
  udiCurrentCycle:                                        UDINT := 1;
  lrLastPos:                                              LREAL;
END_VAR 
VAR // Input variables
  bCylinderDecoupled:                                     BOOL := TRUE;
  uiVentCount:                                            UINT;
  udiERCycles:                                            UDINT;
  udiERTotalCycles:                                       UDINT;
  stERParams:                                             ST_RECIPE_ENDURANCE_RUN;
  stBPDParams:                                            ST_RECIPE_BREAK_PRESSURE;
  stLT1Params:                                            ST_RECIPE_LEAK_TEST1;
  stLT2Params:                                            ST_RECIPE_LEAK_TEST2;
  uiCurrentNokLimitInPercent:                             UINT;
  rCurrentNokDifference:                                  REAL;
  lrStartPos:                                             LREAL;
  sTimer:                                                 STRING;
  rWorkForceATmp:                                         REAL;
  rWorkForceBTmp:                                         REAL;
  rLoadForceATmp:                                         REAL;
  rLoadForceBTmp:                                         REAL;
END_VAR 
VAR
  lrDistanceInM:                                          LREAL;
  lrLastRecordPos:                                        LREAL := 0.0;
  uiRecordDelayCycleCount:                                UINT := 0;
END_VAR 
VAR_TEMP                    	
	iTemp:											                            INT;
END_VAR

// Set FBs and Interfaces ready after switch internal step
IF stSeqCtrlGeneral.iInternalSeqStateCase <> stSeqCtrlGeneral.iLastInternalSeqStateCase AND NOT stSeqCtrlGeneral.bExitSetReadyState THEN
  uiSnippetSeq := uiLastSnippetSeq := 0;
  IF TRUE
  AND itfCounterCyl.M_SetReady()
  AND itfTestCyl.M_SetReady()
  AND itfCounterCylPump.M_SetReady()
  AND itfTestCylPump.M_SetReady()
  AND uiSnippetSeq = 0
  AND uiLastSnippetSeq = 0
  THEN
    stSeqCtrlGeneral.bExitSetReadyState := TRUE;
  ELSE
    RETURN;
  END_IF
END_IF

stSeqCtrlGeneral.strObject:=F_CreateObjectName(strInstancePath);
sTimer := itfTimer.M_GetTimerET(bCustomFormat:= FALSE, sFormat:= '');

// First method call
_m_SequenceManager();
//_m_SaveLastStep();

CASE eSeq OF 
  E_SEQ_VALVE.BASE:;
  
	E_SEQ_PROCESS.INIT: _m_Seq_INIT();
		IF TRUE
		AND (stSeqCtrlGeneral.eActiveSeqState = E_SEQ_GENERAL.DONE) 
		THEN
			eSeq := E_SEQ_PROCESS.BASE;
		END_IF
		
	E_SEQ_PROCESS.SETUP:;
  
	// Process
	E_SEQ_PROCESS.MEASURE_STROKE_LENGTH: _m_Seq_MEASURE_STROKE_LENGTH();
    IF TRUE
		AND stSeqCtrlGeneral.eActiveSeqState = E_SEQ_GENERAL.DONE 
		THEN
			eSeq := E_SEQ_PROCESS.BASE;
		END_IF
  
  E_SEQ_PROCESS.VENT_CYLINDER: _m_Seq_VENT_CYLINDER();
    IF TRUE
		AND stSeqCtrlGeneral.eActiveSeqState = E_SEQ_GENERAL.DONE 
		THEN
			eSeq := E_SEQ_PROCESS.BASE;
		END_IF
  
  E_SEQ_PROCESS.MOVE_TO_SET_POS: _m_Seq_MOVE_TO_SET_POS();
    IF TRUE
		AND stSeqCtrlGeneral.eActiveSeqState = E_SEQ_GENERAL.DONE 
		THEN
			eSeq := E_SEQ_PROCESS.BASE;
		END_IF
  
  E_SEQ_PROCESS.LEAK_TEST_1: _m_Seq_LEAK_TEST_1();
    IF TRUE
		AND stSeqCtrlGeneral.eActiveSeqState = E_SEQ_GENERAL.DONE 
		THEN
			eSeq := E_SEQ_PROCESS.BASE;
		END_IF
  
  E_SEQ_PROCESS.ENDURANCE_RUN: _m_Seq_ENDURANCE_RUN();
    IF TRUE
		AND stSeqCtrlGeneral.eActiveSeqState = E_SEQ_GENERAL.DONE 
		THEN
			eSeq := E_SEQ_PROCESS.BASE;
		END_IF
  
  E_SEQ_PROCESS.STOP_ENGINE: _m_Seq_STOP_ENGINE();
    IF TRUE
		AND stSeqCtrlGeneral.eActiveSeqState = E_SEQ_GENERAL.DONE
		THEN
			eSeq := E_SEQ_PROCESS.BASE;
		END_IF
    
  E_SEQ_PROCESS.STOP: _m_Seq_STOP();
    IF TRUE
		AND stSeqCtrlGeneral.eActiveSeqState = E_SEQ_GENERAL.DONE
		THEN
			eSeq := E_SEQ_PROCESS.BASE;
		END_IF
    
  E_SEQ_PROCESS.RESET_DISTANCE: _m_Seq_RESET_DISTANCE();
    IF TRUE
		AND stSeqCtrlGeneral.eActiveSeqState = E_SEQ_GENERAL.DONE
		THEN
			eSeq := E_SEQ_PROCESS.BASE;
		END_IF
  
  // End
	E_SEQ_PROCESS.END:;
	E_SEQ_PROCESS.ERROR_SEQ:;	
END_CASE

strTemp:=TO_STRING(eSeq);

METHOD PRIVATE _m_DebugManager
VAR_INPUT
	iStepID: int;
END_VAR
IF TRUE
AND THIS^.stSeqCtrlGeneral.bDebugModeActive 
AND NOT THIS^.stSeqCtrlGeneral.bActiveStep
THEN


THIS^.stSeqCtrlGeneral.bBreakpointActive:=FALSE;

FOR i:=0 TO 10 DO
	
	IF TRUE
	AND iStepID=THIS^.stSeqCtrlGeneral.listBreakpoint[i] 
	AND iStepID<>0
	THEN
		EXIT;
	END_IF
END_FOR
IF (i<=10) THEN
	THIS^.stSeqCtrlGeneral.bBreakpointActive:=TRUE;
END_IF

END_IF
END_METHOD

METHOD PRIVATE _m_Delay : BOOL
VAR_INPUT
	DelayTime:	TIME;
END_VAR
THIS^.stSeqCtrlGeneral.bDelayActive:=TRUE;
THIS^.stSeqCtrlGeneral.tDelay:=DelayTime;
_m_Delay:=FALSE;
IF THIS^.stSeqCtrlGeneral.tonDelay.Q THEN
	_m_Delay:=TRUE;
END_IF
END_METHOD

METHOD PRIVATE _m_DistanceRecord : BOOL
VAR_INPUT
END_VAR
// The last position was set at the first call
IF THIS^.uiRecordDelayCycleCount = 0 THEN
  THIS^.lrLastRecordPos := THIS^.itfTestCyl.P_Position;
END_IF

IF THIS^.uiRecordDelayCycleCount >= 100 THEN
THIS^.lrDistanceInM := THIS^.lrDistanceInM + (ABS(THIS^.itfTestCyl.P_Position - THIS^.lrLastRecordPos) / 1000);

THIS^.lrLastRecordPos := THIS^.itfTestCyl.P_Position;
THIS^.uiRecordDelayCycleCount := 1;
END_IF


THIS^.uiRecordDelayCycleCount := THIS^.uiRecordDelayCycleCount + 1;
END_METHOD

METHOD PRIVATE _m_GeneralStepSetting : BOOL
VAR_INPUT
	StepType:			    	E_STEP_STATE_TYPE;
	InfoTextID:					STRING(20);
	EnableDebug:	   			BOOL;	
	
END_VAR
IF THIS^.stSeqCtrlGeneral.bActiveStep THEN
	THIS^.stSeqCtrlGeneral.eStep_Type:=StepType;
	THIS^.stSeqCtrlGeneral.strExtraInfo:= GenLib.F_RET_TXTLIST_ENTRY(strPortNr:='851',strID:='',strTxtLstName:=InfoTextID);
END_IF
END_METHOD

METHOD PRIVATE _m_LeakTest1_LeakDet : BOOL
VAR_INPUT
END_VAR
_m_LeakTest1_LeakDet := THIS^.uiSnippetSeq = 999;

IF TRUE 
AND THIS^.uiSnippetSeq <> THIS^.uiLastSnippetSeq 
THEN
  IF NOT _m_ResetDelayTimer() THEN
    RETURN;
	END_IF
END_IF

THIS^.uiLastSnippetSeq := THIS^.uiSnippetSeq;

CASE THIS^.uiSnippetSeq OF
  0:
    IF TRUE
    AND _m_ResetDelayTimer()
		THEN 
      THIS^.uiSnippetSeq := 10;
		END_IF

  10:
    IF TRUE
    AND _m_Delay(DelayTime:= UINT_TO_TIME(THIS^.uiRecordDelay * 1000))
		THEN 
      THIS^.lrStartPos := THIS^.itfTestCyl.P_Position;
      THIS^.uiSnippetSeq := 20;
		END_IF
  
  20:
    IF TRUE
    AND _m_Delay(DelayTime:= UDINT_TO_TIME(THIS^.stLT1Params.udiDurationPerTest * 60000))
		THEN 
      THIS^.uiSnippetSeq := 999;
		END_IF
    IF ABS(THIS^.lrStartPos - THIS^.itfTestCyl.P_Position) > ABS(THIS^.stLT1Params.rNokLimit) THEN
      THIS^.stSeqCtrlGeneral.iInternalSeqStateCase := 1000; // Abort
		END_IF
    THIS^.rCurrentNokDifference := ABS(THIS^.lrStartPos - THIS^.itfTestCyl.P_Position);
    THIS^.uiCurrentNokLimitInPercent := TO_UINT(100 / ABS(THIS^.stLT1Params.rNokLimit) * THIS^.rCurrentNokDifference);
END_CASE
END_METHOD

METHOD PRIVATE _m_ResetDelayTimer : BOOL
_m_ResetDelayTimer := THIS^.stSeqCtrlGeneral.tonDelay.ET = T#0MS;

THIS^.stSeqCtrlGeneral.tonDelay(IN:= FALSE);
END_METHOD

METHOD PRIVATE _m_SaveLastStep : BOOL
VAR_INPUT
END_VAR
VAR
	i: dint;
END_VAR
IF NOT THIS^.stSeqCtrlGeneral.bActiveStep THEN
	
	FOR i:=49 TO 1 BY -1 DO
			stSeqCtrlGeneral.listLastSteps[i].strStepName:=stSeqCtrlGeneral.listLastSteps[i-1].strStepName;
			stSeqCtrlGeneral.listLastSteps[i].tStepTime:=stSeqCtrlGeneral.listLastSteps[i-1].tStepTime;
			stSeqCtrlGeneral.listLastSteps[i].tDelayTime:=stSeqCtrlGeneral.listLastSteps[i-1].tDelayTime;
	END_FOR
	stSeqCtrlGeneral.listLastSteps[0].strStepName:=TO_STRING(THIS^.eSeq);
	stSeqCtrlGeneral.listLastSteps[1].tStepTime:=THIS^.stSeqCtrlGeneral.tonStepTime.ET;
	stSeqCtrlGeneral.listLastSteps[1].tStepTime:=THIS^.stSeqCtrlGeneral.tonDelay.ET;
ELSE
	stSeqCtrlGeneral.listLastSteps[0].tStepTime:=THIS^.stSeqCtrlGeneral.tonStepTime.ET;
	stSeqCtrlGeneral.listLastSteps[0].tDelayTime:=THIS^.stSeqCtrlGeneral.tonDelay.ET;	
END_IF
END_METHOD

METHOD PRIVATE _m_Seq_ENDURANCE_RUN : E_SEQ_PROCESS
VAR_INPUT
END_VAR
VAR
  ActiveSeq:            STRING;
END_VAR
//THIS^._m_GeneralStepSetting(StepType:=E_STEP_STATE_TYPE.INIT,
ActiveSeq := TO_STRING(THIS^.eSeq);

// Distance record
_m_DistanceRecord();

CASE THIS^.stSeqCtrlGeneral.eActiveSeqState OF
E_SEQ_GENERAL.READY:;

	
E_SEQ_GENERAL.EXECUTE:;
	IF TRUE
	AND _m_Delay(T#1S)
	THEN
		THIS^.stSeqCtrlGeneral.eActiveSeqState := E_SEQ_GENERAL.RESET;
	END_IF
  
E_SEQ_GENERAL.RESET:;
	stSeqCtrlGeneral.iInternalSeqStateCase := 0;
	IF TRUE
	THEN
    THIS^.udiCurrentCycle := 1;
		THIS^.stSeqCtrlGeneral.eActiveSeqState := E_SEQ_GENERAL.BUSY;
	END_IF
  
E_SEQ_GENERAL.BUSY:;
	CASE THIS^.stSeqCtrlGeneral.iInternalSeqStateCase OF
		0: // Check if enable
      IF TRUE
      AND THIS^.bEnable 
      THEN
        THIS^.stSeqCtrlGeneral.iInternalSeqStateCase := 10; 
      ELSE
        THIS^.stSeqCtrlGeneral.iInternalSeqStateCase := 9999; 
			END_IF

    10: // Choice step
      IF TRUE
      AND PrgStation.stRecipeParams.stRecipeEnduranceRun.rSpeedA < THIS^.rMaxSpeedInMmPerSWP * THIS^.rSpeedEfficiencyFactor
      AND PrgStation.stRecipeParams.stRecipeEnduranceRun.rSpeedB < THIS^.rMaxSpeedInMmPerSHP * THIS^.rSpeedEfficiencyFactor
			THEN 
        IF THIS^.udiCurrentCycle > THIS^.udiERCycles THEN
          THIS^.stSeqCtrlGeneral.iInternalSeqStateCase := 1000; 
        ELSE
          THIS^.stSeqCtrlGeneral.iInternalSeqStateCase := 20; 
				END_IF
      ELSE
        THIS^.stSeqCtrlGeneral.iInternalSeqStateCase := 9999;
			END_IF
      
    20: // Add low pressure circuit to counter cylinder
      IF TRUE 
			AND THIS^.itfCounterCyl.M_LowPressureCircuit(bAdd:= TRUE)
			THEN 
				THIS^.stSeqCtrlGeneral.iInternalSeqStateCase := 30; 
			END_IF
      
    30: // Stop
      IF TRUE
      AND _m_Delay(DelayTime:= REAL_TO_TIME(THIS^.stERParams.rDelay * 1000))
      AND THIS^.itfTestCyl.M_Stop()
      AND THIS^.itfCounterCyl.M_Stop()
			THEN 
        THIS^.stSeqCtrlGeneral.iInternalSeqStateCase := 40; 
			END_IF
      
    40: // Move to WP (Max position - 10)
      IF TRUE
      AND THIS^.itfTestCyl.M_ToWP(ePressureType:= E_PRESSURE_TYPE.FORCE, 
                                  rWorkPressure:= THIS^.stERParams.rWorkForceA * 1000, 
                                  bPressureRegulation:= TRUE,
                                  eSpeedType:= E_SPEED_TYPE.MM_PER_SECOND, 
                                  rSpeed:= THIS^.stERParams.rSpeedA)
      AND THIS^.itfCounterCyl.M_ToWP(ePressureType:= E_PRESSURE_TYPE.FORCE, 
                                     rWorkPressure:= THIS^.stERParams.rLoadForceA * 1000, 
                                     bPressureRegulation:= TRUE,
                                     eSpeedType:= E_SPEED_TYPE.PERCENT, 
                                     rSpeed:= 50)
			THEN 
        THIS^.stSeqCtrlGeneral.iInternalSeqStateCase := 41;
			END_IF
      
    41: // Move to WP (Max position - 10)
      IF TRUE
			THEN 
        IF THIS^.itfTestCyl.P_Position >= THIS^.itfTestCyl.P_StrokeLength - ABS(THIS^.stERParams.rTurningPointWP) THEN
				  THIS^.stSeqCtrlGeneral.iInternalSeqStateCase := 50; 
        END_IF
			END_IF
      
    50: // Stop
      IF TRUE
      AND _m_Delay(DelayTime:= REAL_TO_TIME(THIS^.stERParams.rDelay * 1000))
      AND THIS^.itfTestCyl.M_Stop()
      AND THIS^.itfCounterCyl.M_Stop()
			THEN 
        THIS^.stSeqCtrlGeneral.iInternalSeqStateCase := 60; 
			END_IF
      
    60: // Move to HP (Min position + 10)
      IF TRUE
      AND THIS^.bDoubleActing
			THEN 
        THIS^.stSeqCtrlGeneral.iInternalSeqStateCase := 61;
      ELSE
        THIS^.stSeqCtrlGeneral.iInternalSeqStateCase := 62;
			END_IF
      
    61: // Move to HP (Min position + 10)
      IF TRUE
      AND THIS^.itfTestCyl.M_ToHP(ePressureType:= E_PRESSURE_TYPE.FORCE, 
                                  rWorkPressure:= THIS^.stERParams.rWorkForceB * 1000, 
                                  bPressureRegulation:= THIS^.bDoubleActing,
                                  eSpeedType:= E_SPEED_TYPE.MM_PER_SECOND, 
                                  rSpeed:= THIS^.stERParams.rSpeedB)
      AND THIS^.itfCounterCyl.M_ToHP(ePressureType:= E_PRESSURE_TYPE.FORCE, 
                                     rWorkPressure:= THIS^.stERParams.rLoadForceB * 1000, 
                                     bPressureRegulation:= TRUE,
                                     eSpeedType:= E_SPEED_TYPE.PERCENT, 
                                     rSpeed:= 50)
			THEN 
        THIS^.stSeqCtrlGeneral.iInternalSeqStateCase := 70;
			END_IF
      
    62: // Move to HP (Min position + 10)
      IF TRUE
      AND THIS^.itfTestCyl.M_ToHP(ePressureType:= E_PRESSURE_TYPE.VALUE, 
                                  rWorkPressure:= 0, 
                                  bPressureRegulation:= FALSE,
                                  eSpeedType:= E_SPEED_TYPE.MM_PER_SECOND, 
                                  rSpeed:= THIS^.stERParams.rSpeedB)
      AND THIS^.itfCounterCyl.M_ToWP(ePressureType:= E_PRESSURE_TYPE.FORCE, 
                                     rWorkPressure:= THIS^.stERParams.rLoadForceA * 1000, 
                                     bPressureRegulation:= FALSE,
                                     eSpeedType:= E_SPEED_TYPE.PERCENT, 
                                     rSpeed:= 50)
			THEN 
        THIS^.stSeqCtrlGeneral.iInternalSeqStateCase := 70;
			END_IF
      
    70: // Move to HP (Min position + 10)
      IF TRUE
			THEN 
        IF THIS^.itfTestCyl.P_Position <= ABS(THIS^.stERParams.rTurningPointHP) THEN
          THIS^.udiCurrentCycle := THIS^.udiCurrentCycle + 1;
          THIS^.udiERTotalCycles := THIS^.udiERTotalCycles + 1;
				  THIS^.stSeqCtrlGeneral.iInternalSeqStateCase := 10; // Jump backward
        END_IF
			END_IF
      
    1000: // Move to WP (Max position - 10)
      IF TRUE
      AND THIS^.itfTestCyl.M_ToWP(ePressureType:= E_PRESSURE_TYPE.FORCE, 
                                  rWorkPressure:= THIS^.stERParams.rWorkForceA * 1000, 
                                  bPressureRegulation:= TRUE,
                                  eSpeedType:= E_SPEED_TYPE.MM_PER_SECOND, 
                                  rSpeed:= THIS^.stERParams.rSpeedA)
      AND THIS^.itfCounterCyl.M_ToWP( ePressureType:= E_PRESSURE_TYPE.FORCE, 
                                      rWorkPressure:= THIS^.stERParams.rLoadForceA * 1000, 
                                      bPressureRegulation:= TRUE,
                                      eSpeedType:= E_SPEED_TYPE.PERCENT, 
                                      rSpeed:= 50)
			THEN 
        THIS^.stSeqCtrlGeneral.iInternalSeqStateCase := 1010;
			END_IF
      
    1010: // Move to WP (Max position - 10)
      IF TRUE
			THEN 
        IF THIS^.itfTestCyl.P_Position >= THIS^.itfTestCyl.P_StrokeLength / 2 THEN
				  THIS^.stSeqCtrlGeneral.iInternalSeqStateCase := 1020; 
        END_IF
			END_IF
      
    1020: // Exit seq - Disable low pressure circuit
      IF TRUE
      AND _m_Delay(DelayTime:= T#1S)
      AND THIS^.itfCounterCyl.M_LowPressureCircuit(bAdd:= FALSE)
			THEN 
				THIS^.stSeqCtrlGeneral.iInternalSeqStateCase := 1030;
			END_IF
      
    1030: // Exit seq - Stop
      IF TRUE
      AND _m_Delay(DelayTime:= T#1S) 
      AND THIS^.itfTestCyl.M_StopAndLock()
      AND THIS^.itfCounterCyl.M_Stop()
			THEN 
				THIS^.stSeqCtrlGeneral.iInternalSeqStateCase := 1040;
			END_IF
      
    1040: // Set pressure
      IF TRUE 
			AND THIS^.itfCounterCyl.M_SetWorkPressureZero()
      AND THIS^.itfTestCyl.M_SetWorkPressureZero()
			THEN 
				THIS^.stSeqCtrlGeneral.iInternalSeqStateCase := 9999; 
			END_IF
      
	ELSE
		THIS^.stSeqCtrlGeneral.eActiveSeqState := E_SEQ_GENERAL.DONE;  
	END_CASE
	THIS^.stSeqCtrlGeneral.strExtraInfo := CONCAT('Internal state: ', TO_STRING(THIS^.stSeqCtrlGeneral.iInternalSeqStateCase));
E_SEQ_GENERAL.DONE:;
E_SEQ_GENERAL.ERROR:;
E_SEQ_GENERAL.TIME_OUT:; 

IF TRUE
AND THIS^.stSeqCtrlGeneral.bTimeOutActiveQuit 
THEN
  THIS^.stSeqCtrlGeneral.strExtraInfo := 'Bitte quittieren und erneut testen';
  IF TRUE
  //AND itfOpMode.P_QUIT
  THEN
    THIS^.stSeqCtrlGeneral.eActiveSeqState := E_SEQ_GENERAL.EXECUTE;
	END_IF
  
END_IF

ELSE
  THIS^.stSeqCtrlGeneral.eActiveSeqState := E_SEQ_GENERAL.ERROR;
END_CASE
END_METHOD

METHOD PRIVATE _m_Seq_INIT : E_SEQ_PROCESS
VAR_INPUT
END_VAR
VAR
	ActiveSeq: STRING;
END_VAR
VAR
	
END_VAR
//THIS^._m_GeneralStepSetting(StepType:=E_STEP_STATE_TYPE.INIT,
ActiveSeq := TO_STRING(THIS^.eSeq);

CASE THIS^.stSeqCtrlGeneral.eActiveSeqState OF
E_SEQ_GENERAL.READY:;

	
E_SEQ_GENERAL.EXECUTE:;
	IF TRUE
	THEN
		THIS^.stSeqCtrlGeneral.eActiveSeqState := E_SEQ_GENERAL.RESET;
	END_IF
  
E_SEQ_GENERAL.RESET:;
	stSeqCtrlGeneral.iInternalSeqStateCase := 0;
	IF TRUE
	THEN
    THIS^.udiERTotalCycles := 0;
		THIS^.stSeqCtrlGeneral.eActiveSeqState := E_SEQ_GENERAL.BUSY;
	END_IF
  
E_SEQ_GENERAL.BUSY:;
	CASE THIS^.stSeqCtrlGeneral.iInternalSeqStateCase OF
		0:  // Switch off the counter cylinder pump
      IF TRUE 
			//AND THIS^.itfCounterCylPump.M_Off()
			THEN 
				THIS^.stSeqCtrlGeneral.iInternalSeqStateCase := 10; 
			END_IF
      
    10: // Enable bypass
      IF TRUE 
			AND THIS^.itfCounterCylPump.M_Bypass(bEnable:= TRUE)
			THEN 
				THIS^.stSeqCtrlGeneral.iInternalSeqStateCase := 20; 
			END_IF
      
    20: // Switch off the test cylinder pump
      IF TRUE 
			//AND THIS^.itfTestCylPump.M_Off()
			THEN 
				THIS^.stSeqCtrlGeneral.iInternalSeqStateCase := 30; 
			END_IF
      
		30:	// Reset counter cylinder
      IF TRUE 
			AND THIS^.itfCounterCyl.M_Reset()
			THEN 
				THIS^.stSeqCtrlGeneral.iInternalSeqStateCase := 40; 
			END_IF
      
		40: // Reset test cylinder
      IF TRUE 
			AND THIS^.itfTestCyl.M_Reset()
			THEN 
				THIS^.stSeqCtrlGeneral.iInternalSeqStateCase := 50; 
			END_IF
      
		50: // Turn on the counter cylinder pump
      IF TRUE 
			AND THIS^.itfCounterCylPump.M_On() 
			THEN 
				THIS^.stSeqCtrlGeneral.iInternalSeqStateCase := 60; 
			END_IF
      
		60:	// Turn on the test cylinder pump
      IF TRUE 
			AND THIS^.itfTestCylPump.M_On()
			THEN 
				THIS^.stSeqCtrlGeneral.iInternalSeqStateCase := 1000; 
			END_IF
      
    1000: // Exit step
      IF TRUE
			THEN 
				THIS^.stSeqCtrlGeneral.iInternalSeqStateCase := 9999;
			END_IF
      
	ELSE
		THIS^.stSeqCtrlGeneral.eActiveSeqState := E_SEQ_GENERAL.DONE;  
	END_CASE
	THIS^.stSeqCtrlGeneral.strExtraInfo := CONCAT('Internal state: ', TO_STRING(THIS^.stSeqCtrlGeneral.iInternalSeqStateCase));
E_SEQ_GENERAL.DONE:;
E_SEQ_GENERAL.ERROR:;
E_SEQ_GENERAL.TIME_OUT:; 

IF TRUE
AND THIS^.stSeqCtrlGeneral.bTimeOutActiveQuit 
THEN
  THIS^.stSeqCtrlGeneral.strExtraInfo := 'Bitte quittieren und erneut testen';
  IF TRUE
  //AND itfOpMode.P_QUIT
  THEN
    THIS^.stSeqCtrlGeneral.eActiveSeqState := E_SEQ_GENERAL.EXECUTE;
	END_IF
  
END_IF

ELSE
  THIS^.stSeqCtrlGeneral.eActiveSeqState := E_SEQ_GENERAL.ERROR;
END_CASE
END_METHOD

METHOD PRIVATE _m_Seq_LEAK_TEST_1 : E_SEQ_PROCESS
VAR_INPUT
END_VAR
VAR
  ActiveSeq: STRING;
END_VAR
//THIS^._m_GeneralStepSetting(StepType:=E_STEP_STATE_TYPE.INIT,
ActiveSeq := TO_STRING(THIS^.eSeq);

// Distance record
_m_DistanceRecord();

CASE THIS^.stSeqCtrlGeneral.eActiveSeqState OF
E_SEQ_GENERAL.READY:;

	
E_SEQ_GENERAL.EXECUTE:;
	IF TRUE
	AND _m_Delay(T#1S)
	THEN
		THIS^.stSeqCtrlGeneral.eActiveSeqState := E_SEQ_GENERAL.RESET;
	END_IF
  
E_SEQ_GENERAL.RESET:;
	stSeqCtrlGeneral.iInternalSeqStateCase := 0;
	IF TRUE
	THEN
		THIS^.stSeqCtrlGeneral.eActiveSeqState := E_SEQ_GENERAL.BUSY;
	END_IF
  
E_SEQ_GENERAL.BUSY:;
	CASE THIS^.stSeqCtrlGeneral.iInternalSeqStateCase OF
		0: // Check if enable
      IF TRUE
      AND THIS^.bEnable 
      THEN
        THIS^.stSeqCtrlGeneral.iInternalSeqStateCase := 10; 
      ELSE
        THIS^.stSeqCtrlGeneral.iInternalSeqStateCase := 9999; 
			END_IF

    10: // Shut off low pressure circuit to counter cylinder and switch off pump
      IF TRUE
      AND THIS^.itfCounterCyl.M_LowPressureCircuit(bAdd:= FALSE)
			THEN 
        IF THIS^.bDoubleActing THEN
				  THIS^.stSeqCtrlGeneral.iInternalSeqStateCase := 20; 
        ELSE
          THIS^.stSeqCtrlGeneral.iInternalSeqStateCase := 21; 
        END_IF
			END_IF
      
    20: // Move to HP (Min position + 10mm)
      IF TRUE
      AND THIS^.itfTestCyl.M_ToHP(ePressureType:= E_PRESSURE_TYPE.FORCE, 
                                  rWorkPressure:= THIS^.stLT1Params.rLoadForceB * 1000, 
                                  bPressureRegulation:= FALSE,
                                  eSpeedType:= E_SPEED_TYPE.PERCENT, 
                                  rSpeed:= 50)
      AND THIS^.itfCounterCyl.M_ToHP(ePressureType:= E_PRESSURE_TYPE.VALUE, 
                                     rWorkPressure:= 0, 
                                     bPressureRegulation:= FALSE,
                                     eSpeedType:= E_SPEED_TYPE.PERCENT, 
                                     rSpeed:= 50)
			THEN 
        IF THIS^.itfTestCyl.P_Position <= ABS(THIS^.stLT1Params.rDistanceBeforeEndPosHP) THEN
				  THIS^.stSeqCtrlGeneral.iInternalSeqStateCase := 30; 
        END_IF
			END_IF
      
    21: // Move to HP (Min position + 10mm)
      IF TRUE
      AND THIS^.itfTestCyl.M_ToHP(ePressureType:= E_PRESSURE_TYPE.VALUE, 
                                  rWorkPressure:= 0, 
                                  bPressureRegulation:= FALSE,
                                  eSpeedType:= E_SPEED_TYPE.PERCENT, 
                                  rSpeed:= 50)
      AND THIS^.itfCounterCyl.M_ToWP(ePressureType:= E_PRESSURE_TYPE.FORCE, 
                                     rWorkPressure:= THIS^.stLT1Params.rLoadForceA * 1000, 
                                     bPressureRegulation:= FALSE,
                                     eSpeedType:= E_SPEED_TYPE.PERCENT, 
                                     rSpeed:= 50)
			THEN 
        IF THIS^.itfTestCyl.P_Position <= ABS(THIS^.stLT1Params.rDistanceBeforeEndPosHP) THEN
				  THIS^.stSeqCtrlGeneral.iInternalSeqStateCase := 30; 
        END_IF
			END_IF
      
    30: // Stop and lock
      IF TRUE
      AND _m_Delay(DelayTime:= T#1S)
      AND THIS^.itfTestCyl.M_StopAndLock()
      AND THIS^.itfCounterCyl.M_Stop()
			THEN 
        THIS^.stSeqCtrlGeneral.iInternalSeqStateCase := 40; 
			END_IF
      
    40: // Set cylinder pressure to 0
      IF TRUE
      AND THIS^.itfTestCyl.M_SetWorkPressureZero()
			THEN 
        THIS^.stSeqCtrlGeneral.iInternalSeqStateCase := 50; 
			END_IF
      
    50: // Start leak test push (HP endposition + 10mm)
      IF TRUE
      AND _m_Delay(DelayTime:= T#1S)
      AND THIS^.itfCounterCyl.M_ToWP(ePressureType:= E_PRESSURE_TYPE.FORCE, 
                                     rWorkPressure:= THIS^.stLT1Params.rLoadForceA * 1000, 
                                     bPressureRegulation:= TRUE,
                                     eSpeedType:= E_SPEED_TYPE.PERCENT, 
                                     rSpeed:= 100)
			THEN 
        THIS^.stSeqCtrlGeneral.iInternalSeqStateCase := 60;
			END_IF
      
    60: // Leak detection
      IF TRUE
      AND _m_LeakTest1_LeakDet()
			THEN 
        THIS^.stSeqCtrlGeneral.iInternalSeqStateCase := 70;
			END_IF
      
